C07289=1017.873,162.387,378.674,167.472,52.697,159.777
C07290=1017.878,162.636,378.653,167.475,52.688,159.776
C07291=1017.882,162.885,378.632,167.480,52.680,159.775
C07292=1017.887,163.133,378.611,167.483,52.671,159.774
C07293=1017.892,163.383,378.590,167.486,52.662,159.772
C07294=1017.897,163.632,378.569,167.490,52.654,159.772
C07295=1017.902,163.881,378.548,167.494,52.645,159.771
C07296=1017.906,164.131,378.527,167.498,52.637,159.770
C07297=1017.911,164.379,378.507,167.501,52.628,159.768
C07298=1017.916,164.628,378.485,167.504,52.619,159.767
C07299=1017.921,164.877,378.465,167.508,52.611,159.766
C07300=1017.925,165.127,378.443,167.512,52.602,159.765
C07301=1017.930,165.376,378.422,167.516,52.593,159.764
C07302=1017.935,165.625,378.402,167.519,52.585,159.763
C07303=1017.939,165.873,378.380,167.523,52.575,159.762
C07304=1017.945,166.122,378.360,167.527,52.567,159.761
C07305=1017.949,166.372,378.338,167.530,52.558,159.760
C07306=1017.954,166.621,378.317,167.534,52.550,159.759
C07307=1017.959,166.870,378.296,167.538,52.541,159.758
C07308=1017.964,167.119,378.275,167.542,52.532,159.757
C07309=1017.969,167.368,378.254,167.545,52.524,159.756
C07310=1017.974,167.618,378.233,167.548,52.515,159.755
C07311=1017.978,167.866,378.212,167.553,52.506,159.754
C07312=1017.983,168.115,378.191,167.556,52.498,159.753
C07313=1017.988,168.364,378.170,167.560,52.489,159.752
C07314=1017.993,168.613,378.149,167.564,52.480,159.751
C07315=1017.998,168.862,378.128,167.568,52.472,159.750
C07316=1018.002,169.112,378.106,167.571,52.463,159.749
C07317=1018.008,169.360,378.085,167.575,52.454,159.748
C07318=1018.012,169.610,378.064,167.579,52.446,159.747
C07319=1018.017,169.859,378.043,167.582,52.437,159.746
C07320=1018.022,170.108,378.022,167.587,52.429,159.745
C07321=1018.027,170.357,378.000,167.590,52.420,159.744
C07322=1018.032,170.606,377.980,167.594,52.411,159.743
C07323=1018.038,170.887,377.956,167.598,52.401,159.742
C07324=1018.043,171.168,377.932,167.603,52.392,159.741
C07325=1018.048,171.449,377.908,167.607,52.382,159.739
C07326=1018.054,171.731,377.884,167.611,52.372,159.738
C07327=1018.058,171.980,377.863,167.615,52.364,159.737
C07328=1018.064,172.228,377.842,167.618,52.355,159.736
C07329=1018.069,172.478,377.820,167.623,52.346,159.735
C07330=1018.074,172.727,377.799,167.627,52.338,159.734
C07331=1018.079,172.976,377.778,167.630,52.329,159.733
C07332=1018.084,173.225,377.756,167.634,52.320,159.732
C07333=1018.089,173.474,377.735,167.638,52.312,159.731
C07334=1018.094,173.723,377.713,167.642,52.302,159.730
C07335=1018.098,173.972,377.692,167.645,52.294,159.729
C07336=1018.104,174.221,377.671,167.649,52.286,159.728
C07337=1018.108,174.470,377.650,167.654,52.276,159.727
C07338=1018.114,174.719,377.629,167.657,52.268,159.726
C07339=1018.118,174.968,377.607,167.662,52.259,159.725
C07340=1018.123,175.217,377.586,167.665,52.250,159.724
C07341=1018.129,175.466,377.565,167.669,52.241,159.723
C07342=1018.133,175.715,377.543,167.673,52.233,159.722
C07343=1018.138,175.964,377.522,167.676,52.225,159.721
C07344=1018.143,176.213,377.501,167.681,52.215,159.720
C07345=1018.148,176.462,377.479,167.684,52.207,159.719
C07346=1018.154,176.711,377.458,167.689,52.198,159.718
C07347=1018.159,176.960,377.436,167.692,52.190,159.717
C07348=1018.163,177.210,377.415,167.697,52.181,159.716
C07349=1018.169,177.458,377.394,167.700,52.172,159.715
C07350=1018.174,177.707,377.372,167.705,52.164,159.714
C07351=1018.178,177.956,377.351,167.708,52.155,159.713
C07352=1018.184,178.205,377.329,167.713,52.146,159.712
C07353=1018.189,178.454,377.307,167.716,52.138,159.711
C07354=1018.194,178.704,377.286,167.721,52.129,159.710
C07355=1018.199,178.952,377.265,167.724,52.120,159.709
C07356=1018.204,179.201,377.243,167.729,52.112,159.708
C07357=1018.210,179.450,377.222,167.732,52.103,159.707
C07358=1018.214,179.699,377.200,167.737,52.094,159.706
C07359=1018.220,179.949,377.178,167.740,52.086,159.705
C07360=1018.225,180.198,377.158,167.745,52.077,159.704
C07361=1018.230,180.447,377.136,167.748,52.068,159.703
C07362=1018.235,180.695,377.114,167.753,52.060,159.702
C07363=1018.240,180.944,377.093,167.756,52.051,159.701
C07364=1018.245,181.194,377.071,167.761,52.042,159.700
C07365=1018.250,181.443,377.049,167.764,52.034,159.699
C07366=1018.256,181.691,377.028,167.769,52.025,159.698
C07367=1018.261,181.940,377.006,167.772,52.016,159.697
C07368=1018.266,182.190,376.984,167.777,52.008,159.696
C07369=1018.270,182.439,376.961,167.781,52.000,159.695
C07370=1018.275,182.688,376.940,167.785,51.991,159.694
C07371=1018.280,182.937,376.918,167.789,51.983,159.693
C07372=1018.284,183.186,376.895,167.793,51.975,159.692
C07373=1018.289,183.435,376.873,167.797,51.965,159.691
C07374=1018.294,183.684,376.851,167.801,51.957,159.690
C07375=1018.299,183.933,376.829,167.805,51.949,159.689
C07376=1018.303,184.182,376.807,167.809,51.941,159.688
C07377=1018.309,184.431,376.784,167.813,51.932,159.687
C07378=1018.314,184.680,376.762,167.818,51.924,159.686
C07379=1018.318,184.928,376.740,167.821,51.916,159.685
C07380=1018.322,185.178,376.718,167.825,51.907,159.684
C07381=1018.328,185.427,376.695,167.830,51.899,159.684
C07382=1018.333,185.675,376.673,167.833,51.891,159.683
C07383=1018.337,185.924,376.650,167.838,51.882,159.682
C07384=1018.342,186.173,376.629,167.842,51.874,159.681
C07385=1018.347,186.423,376.606,167.846,51.865,159.680
C07386=1018.351,186.672,376.584,167.850,51.857,159.679
C07387=1018.357,186.952,376.559,167.854,51.848,159.678
C07388=1018.363,187.233,376.533,167.860,51.838,159.677
C07389=1018.368,187.514,376.508,167.864,51.829,159.676
C07390=1018.374,187.794,376.483,167.869,51.819,159.675
C07391=1018.379,188.044,376.461,167.872,51.811,159.674
C07392=1018.384,188.292,376.439,167.877,51.802,159.673
C07393=1018.388,188.541,376.416,167.881,51.794,159.672
C07394=1018.394,188.790,376.393,167.886,51.785,159.671
C07395=1018.398,189.039,376.371,167.889,51.777,159.670
C07396=1018.403,189.288,376.348,167.894,51.769,159.669
C07397=1018.408,189.537,376.326,167.898,51.761,159.668
C07398=1018.413,189.786,376.304,167.903,51.752,159.667
C07399=1018.419,190.035,376.281,167.906,51.744,159.666
C07400=1018.423,190.284,376.259,167.911,51.736,159.665
C07401=1018.428,190.533,376.237,167.915,51.727,159.664
C07402=1018.433,190.782,376.214,167.919,51.719,159.663
C07403=1018.438,191.031,376.192,167.923,51.711,159.662
C07404=1018.443,191.280,376.169,167.928,51.702,159.661
C07405=1018.448,191.529,376.147,167.932,51.694,159.661
C07406=1018.453,191.777,376.124,167.936,51.685,159.660
C07407=1018.458,192.027,376.101,167.940,51.677,159.659
C07408=1018.463,192.275,376.079,167.945,51.668,159.658
C07409=1018.468,192.525,376.056,167.949,51.660,159.657
C07410=1018.473,192.773,376.034,167.953,51.651,159.656
C07411=1018.478,193.022,376.011,167.958,51.643,159.655
C07412=1018.483,193.271,375.989,167.962,51.635,159.654
C07413=1018.488,193.520,375.966,167.967,51.627,159.653
C07414=1018.493,193.769,375.944,167.970,51.618,159.652
C07415=1018.498,194.017,375.921,167.975,51.610,159.651
C07416=1018.503,194.267,375.898,167.980,51.602,159.651
C07417=1018.508,194.515,375.876,167.983,51.593,159.649
C07418=1018.514,194.764,375.853,167.988,51.585,159.649
C07419=1018.518,195.014,375.830,167.992,51.577,159.648
C07420=1018.523,195.262,375.808,167.996,51.568,159.647
C07421=1018.529,195.512,375.785,168.001,51.559,159.646
C07422=1018.533,195.760,375.762,168.005,51.551,159.645
C07423=1018.539,196.009,375.739,168.010,51.543,159.644
C07424=1018.544,196.258,375.717,168.013,51.535,159.643
C07425=1018.549,196.507,375.694,168.018,51.526,159.642
C07426=1018.554,196.756,375.672,168.023,51.518,159.641
C07427=1018.559,197.005,375.649,168.027,51.509,159.640
C07428=1018.564,197.253,375.626,168.032,51.501,159.639
C07429=1018.569,197.503,375.604,168.036,51.493,159.639
C07430=1018.575,197.752,375.581,168.040,51.485,159.638
C07431=1018.580,198.000,375.558,168.045,51.476,159.637
C07432=1018.585,198.249,375.534,168.050,51.468,159.636
C07433=1018.590,198.498,375.513,168.054,51.460,159.635
C07434=1018.596,198.747,375.490,168.058,51.451,159.634
C07435=1018.601,198.996,375.466,168.063,51.442,159.633
C07436=1018.605,199.245,375.444,168.068,51.434,159.632
C07437=1018.610,199.494,375.421,168.072,51.426,159.631
C07438=1018.616,199.743,375.398,168.077,51.418,159.630
C07439=1018.621,199.992,375.375,168.081,51.410,159.630
C07440=1018.625,200.241,375.351,168.085,51.402,159.629
C07441=1018.631,200.490,375.328,168.090,51.393,159.628
C07442=1018.636,200.738,375.305,168.094,51.385,159.627
C07443=1018.641,200.987,375.281,168.099,51.377,159.626
C07444=1018.645,201.236,375.258,168.103,51.369,159.625
C07445=1018.651,201.485,375.235,168.108,51.361,159.624
C07446=1018.656,201.734,375.212,168.112,51.352,159.623
C07447=1018.660,201.983,375.189,168.116,51.344,159.622
C07448=1018.666,202.231,375.166,168.121,51.336,159.622
C07449=1018.671,202.481,375.142,168.126,51.328,159.621
C07450=1018.675,202.729,375.119,168.130,51.320,159.620
C07451=1018.702,203.979,375.000,168.600,51.411,159.725
C07452=1018.707,204.207,374.977,168.603,51.404,159.724
C07453=1018.713,204.434,374.955,168.607,51.398,159.723
C07454=1018.718,204.661,374.932,168.610,51.391,159.723
C07455=1018.724,204.888,374.910,168.614,51.385,159.722
C07456=1018.730,205.116,374.887,168.617,51.378,159.721
C07457=1018.735,205.343,374.863,168.620,51.372,159.720
C07458=1018.740,205.570,374.841,168.624,51.365,159.720
C07459=1018.747,205.819,374.816,168.628,51.358,159.719
C07460=1018.753,206.068,374.791,168.631,51.351,159.718
C07461=1018.758,206.316,374.766,168.635,51.343,159.717
C07462=1018.764,206.565,374.741,168.640,51.336,159.716
C07463=1018.771,206.813,374.716,168.643,51.329,159.715
C07464=1018.777,207.062,374.690,168.647,51.322,159.715
C07465=1018.782,207.311,374.666,168.650,51.315,159.714
C07466=1018.788,207.559,374.641,168.655,51.308,159.713
C07467=1018.794,207.808,374.615,168.658,51.301,159.712
C07468=1018.801,208.057,374.590,168.662,51.294,159.711
C07469=1018.806,208.305,374.565,168.666,51.287,159.711
C07470=1018.812,208.554,374.540,168.670,51.280,159.710
C07471=1018.818,208.803,374.515,168.674,51.273,159.709
C07472=1018.824,209.052,374.489,168.677,51.266,159.708
C07473=1018.830,209.300,374.464,168.682,51.260,159.707
C07474=1018.836,209.548,374.439,168.685,51.253,159.707
C07475=1018.842,209.797,374.414,168.689,51.246,159.706
C07476=1018.848,210.046,374.388,168.692,51.239,159.705
C07477=1018.854,210.294,374.363,168.697,51.232,159.704
C07478=1018.860,210.543,374.337,168.700,51.225,159.703
C07479=1018.866,210.792,374.312,168.705,51.218,159.703
C07480=1018.872,211.040,374.287,168.708,51.212,159.702
C07481=1018.878,211.289,374.261,168.712,51.204,159.701
C07482=1018.883,211.538,374.235,168.715,51.198,159.700
C07483=1018.889,211.786,374.210,168.720,51.191,159.700
C07484=1018.896,212.035,374.185,168.723,51.184,159.699
C07485=1018.901,212.284,374.159,168.728,51.177,159.698
C07486=1018.907,212.533,374.133,168.731,51.170,159.697
C07487=1018.913,212.781,374.108,168.735,51.164,159.696
C07488=1018.919,213.029,374.083,168.739,51.157,159.696
C07489=1018.925,213.278,374.057,168.742,51.150,159.695
C07490=1018.931,213.527,374.032,168.747,51.144,159.694
C07491=1018.937,213.775,374.006,168.750,51.137,159.693
C07492=1018.942,214.024,373.981,168.754,51.130,159.693
C07493=1018.949,214.273,373.955,168.758,51.124,159.692
C07494=1018.955,214.521,373.929,168.762,51.117,159.691
C07495=1018.961,214.770,373.904,168.765,51.110,159.690
C07496=1018.967,215.019,373.878,168.770,51.103,159.690
C07497=1018.973,215.268,373.853,168.773,51.096,159.689
C07498=1018.979,215.516,373.827,168.777,51.090,159.688
C07499=1018.984,215.764,373.802,168.781,51.083,159.687
C07500=1018.990,216.013,373.776,168.785,51.076,159.687
C07501=1018.997,216.261,373.750,168.789,51.070,159.686
C07502=1019.003,216.510,373.725,168.793,51.063,159.685
C07503=1019.009,216.759,373.699,168.797,51.057,159.685
C07504=1019.015,217.007,373.674,168.801,51.050,159.684
C07505=1019.021,217.256,373.648,168.805,51.043,159.683
C07506=1019.027,217.505,373.622,168.809,51.037,159.682
C07507=1019.033,217.753,373.596,168.812,51.031,159.682
C07508=1019.039,218.002,373.571,168.816,51.023,159.681
C07509=1019.046,218.250,373.545,168.820,51.017,159.680
C07510=1019.051,218.499,373.519,168.824,51.010,159.679
C07511=1019.057,218.726,373.495,168.827,51.004,159.679
C07512=1019.062,218.955,373.472,168.831,50.999,159.678
C07513=1019.068,219.183,373.448,168.835,50.993,159.677
C07514=1019.073,219.411,373.423,168.839,50.987,159.677
C07515=1019.078,219.639,373.400,168.842,50.981,159.676
C07516=1019.084,219.867,373.376,168.846,50.975,159.676
C07517=1019.089,220.095,373.352,168.849,50.969,159.675
C07518=1019.095,220.322,373.328,168.853,50.963,159.674
C07519=1019.100,220.571,373.302,168.856,50.957,159.674
C07520=1019.107,220.819,373.276,168.861,50.950,159.673
C07521=1019.112,221.068,373.250,168.864,50.944,159.672
C07522=1019.118,221.317,373.223,168.868,50.938,159.671
C07523=1019.124,221.565,373.198,168.873,50.931,159.671
C07524=1019.131,221.814,373.171,168.876,50.925,159.670
C07525=1019.137,222.063,373.146,168.880,50.919,159.669
C07526=1019.143,222.311,373.119,168.884,50.912,159.669
C07527=1019.148,222.560,373.093,168.888,50.906,159.668
C07528=1019.155,222.808,373.067,168.892,50.900,159.667
C07529=1019.160,223.057,373.041,168.897,50.894,159.667
C07530=1019.167,223.305,373.015,168.900,50.887,159.666
C07531=1019.172,223.554,372.988,168.904,50.881,159.665
C07532=1019.178,223.803,372.962,168.908,50.874,159.665
C07533=1019.185,224.052,372.936,168.912,50.868,159.664
C07534=1019.190,224.300,372.910,168.916,50.862,159.663
C07535=1019.197,224.549,372.884,168.920,50.856,159.663
C07536=1019.203,224.797,372.857,168.924,50.850,159.662
C07537=1019.208,225.046,372.832,168.928,50.843,159.662
C07538=1019.215,225.294,372.805,168.932,50.836,159.661
C07539=1019.220,225.542,372.779,168.936,50.830,159.660
C07540=1019.227,225.792,372.753,168.940,50.824,159.659
C07541=1019.233,226.040,372.726,168.944,50.818,159.659
C07542=1019.239,226.288,372.700,168.948,50.812,159.658
C07543=1019.245,226.536,372.674,168.952,50.806,159.658
C07544=1019.251,226.785,372.648,168.955,50.800,159.657
C07545=1019.257,227.034,372.621,168.960,50.793,159.656
C07546=1019.263,227.283,372.594,168.964,50.787,159.656
C07547=1019.269,227.531,372.568,168.967,50.781,159.655
C07548=1019.275,227.779,372.541,168.972,50.776,159.655
C07549=1019.281,228.028,372.515,168.976,50.769,159.654
C07550=1019.287,228.276,372.488,168.980,50.763,159.653
C07551=1019.293,228.526,372.462,168.984,50.757,159.653
C07552=1019.299,228.774,372.435,168.987,50.751,159.652
C07553=1019.305,229.022,372.409,168.992,50.745,159.651
C07554=1019.311,229.270,372.383,168.996,50.738,159.651
C07555=1019.317,229.519,372.355,169.000,50.733,159.650
C07556=1019.323,229.768,372.329,169.004,50.727,159.650
C07557=1019.329,230.016,372.302,169.007,50.721,159.649
C07558=1019.335,230.265,372.276,169.012,50.715,159.648
C07559=1019.341,230.514,372.249,169.016,50.709,159.648
C07560=1019.347,230.762,372.222,169.020,50.703,159.647
C07561=1019.353,231.010,372.195,169.024,50.697,159.647
C07562=1019.358,231.259,372.169,169.028,50.692,159.646
C07563=1019.365,231.508,372.142,169.033,50.685,159.646
C07564=1019.371,231.755,372.114,169.036,50.679,159.645
C07565=1019.377,232.004,372.088,169.040,50.674,159.644
C07566=1019.383,232.253,372.061,169.044,50.668,159.644
C07567=1019.389,232.501,372.034,169.048,50.662,159.643
C07568=1019.394,232.750,372.007,169.053,50.656,159.643
C07569=1019.400,232.998,371.981,169.057,50.650,159.642
C07570=1019.407,233.247,371.954,169.060,50.644,159.641
C07571=1019.412,233.470,371.929,169.064,50.639,159.641
C07572=1019.418,233.695,371.905,169.068,50.633,159.640
C07573=1019.423,233.918,371.881,169.072,50.628,159.640
C07574=1019.429,234.143,371.857,169.075,50.623,159.639
C07575=1019.434,234.366,371.833,169.079,50.618,159.639
C07576=1019.440,234.590,371.808,169.082,50.613,159.638
C07577=1019.445,234.814,371.784,169.086,50.607,159.638
C07578=1019.450,235.038,371.759,169.089,50.602,159.637
C07579=1019.456,235.286,371.732,169.094,50.596,159.637
C07580=1019.462,235.534,371.706,169.098,50.590,159.636
C07581=1019.468,235.783,371.678,169.102,50.585,159.636
C07582=1019.474,236.031,371.651,169.106,50.579,159.635
C07583=1019.481,236.280,371.624,169.110,50.574,159.635
C07584=1019.487,236.528,371.597,169.114,50.568,159.634
C07585=1019.492,236.776,371.570,169.119,50.562,159.634
C07586=1019.499,237.025,371.543,169.123,50.556,159.633
C07587=1019.505,237.273,371.516,169.127,50.551,159.632
C07588=1019.511,237.522,371.489,169.131,50.545,159.632
C07589=1019.517,237.771,371.462,169.135,50.539,159.631
C07590=1019.524,238.019,371.434,169.139,50.534,159.631
C07591=1019.529,238.267,371.408,169.144,50.527,159.630
C07592=1019.535,238.516,371.381,169.148,50.522,159.630
C07593=1019.541,238.765,371.353,169.152,50.517,159.629
C07594=1019.547,239.013,371.326,169.156,50.511,159.629
C07595=1019.554,239.261,371.298,169.160,50.505,159.628
C07596=1019.559,239.510,371.272,169.164,50.500,159.628
C07597=1019.565,239.758,371.244,169.168,50.495,159.627
C07598=1019.571,240.007,371.217,169.172,50.489,159.627
C07599=1019.578,240.255,371.189,169.176,50.483,159.626
C07600=1019.583,240.503,371.161,169.180,50.478,159.626
C07601=1019.590,240.752,371.134,169.185,50.472,159.625
C07602=1019.596,241.000,371.107,169.189,50.467,159.625
C07603=1019.602,241.249,371.078,169.194,50.461,159.624
C07604=1019.607,241.497,371.052,169.197,50.455,159.624
C07605=1019.614,241.746,371.024,169.201,50.450,159.623
C07606=1019.619,241.994,370.996,169.206,50.445,159.623
C07607=1019.626,242.243,370.969,169.210,50.439,159.622
C07608=1019.632,242.491,370.942,169.214,50.434,159.622
C07609=1019.638,242.739,370.913,169.218,50.429,159.621
C07610=1019.644,242.988,370.887,169.222,50.423,159.621
C07611=1019.650,243.236,370.859,169.226,50.418,159.620
C07612=1019.656,243.484,370.831,169.230,50.413,159.620
C07613=1019.661,243.733,370.803,169.235,50.407,159.620
C07614=1019.668,243.981,370.775,169.239,50.402,159.619
C07615=1019.673,244.230,370.748,169.243,50.397,159.619
C07616=1019.679,244.478,370.720,169.247,50.391,159.618
C07617=1019.685,244.726,370.692,169.251,50.386,159.618
C07618=1019.691,244.975,370.664,169.255,50.381,159.617
C07619=1019.697,245.223,370.636,169.259,50.375,159.617
C07620=1019.703,245.472,370.608,169.264,50.370,159.616
C07621=1019.709,245.720,370.580,169.268,50.365,159.616
C07622=1019.715,245.968,370.552,169.272,50.360,159.616
C07623=1019.721,246.217,370.524,169.276,50.355,159.615
C07624=1019.726,246.465,370.496,169.280,50.349,159.615
C07625=1019.733,246.713,370.468,169.285,50.344,159.614
C07626=1019.739,246.962,370.440,169.289,50.339,159.614
C07627=1019.744,247.210,370.412,169.293,50.334,159.613
C07628=1019.751,247.459,370.384,169.297,50.329,159.613
C07629=1019.756,247.707,370.356,169.302,50.323,159.612
C07630=1019.762,247.956,370.328,169.307,50.318,159.612
C07631=1019.768,248.176,370.304,169.310,50.313,159.612
C07632=1019.773,248.397,370.278,169.314,50.309,159.611
C07633=1019.779,248.617,370.254,169.318,50.304,159.611
C07634=1019.784,248.838,370.229,169.321,50.299,159.610
C07635=1019.790,249.059,370.204,169.325,50.295,159.610
C07636=1019.794,249.279,370.179,169.330,50.290,159.610
C07637=1019.801,249.500,370.154,169.333,50.286,159.610
C07638=1019.805,249.721,370.129,169.337,50.282,159.609
C07639=1019.812,249.968,370.101,169.341,50.276,159.609
C07640=1019.818,250.216,370.073,169.345,50.271,159.608
C07641=1019.824,250.465,370.044,169.349,50.266,159.608
C07642=1019.830,250.714,370.017,169.354,50.261,159.607
C07643=1019.836,250.962,369.988,169.358,50.256,159.607
C07644=1019.842,251.210,369.960,169.362,50.251,159.607
C07645=1019.849,251.458,369.932,169.366,50.246,159.606
C07646=1019.854,251.707,369.904,169.371,50.240,159.606
C07647=1019.860,251.956,369.875,169.375,50.236,159.606
C07648=1019.867,252.204,369.848,169.379,50.230,159.605
C07649=1019.873,252.452,369.819,169.384,50.226,159.605
C07650=1019.879,252.700,369.790,169.388,50.220,159.604
C07651=1019.885,252.949,369.763,169.392,50.215,159.604
C07652=1019.891,253.198,369.734,169.397,50.210,159.604
C07653=1019.897,253.445,369.706,169.401,50.205,159.603
C07654=1019.904,253.694,369.678,169.405,50.200,159.603
C07655=1019.910,253.942,369.650,169.410,50.195,159.602
C07656=1019.916,254.190,369.621,169.414,50.191,159.602
C07657=1019.923,254.439,369.593,169.418,50.185,159.602
C07658=1019.928,254.688,369.565,169.423,50.181,159.601
C07659=1019.934,254.935,369.536,169.427,50.175,159.601
C07660=1019.941,255.183,369.508,169.431,50.171,159.601
C07661=1019.947,255.432,369.480,169.436,50.165,159.600
C07662=1019.953,255.680,369.451,169.440,50.161,159.600
C07663=1019.960,255.929,369.423,169.444,50.155,159.599
C07664=1019.966,256.177,369.394,169.449,50.151,159.599
C07665=1019.972,256.426,369.366,169.453,50.145,159.599
C07666=1019.979,256.673,369.337,169.458,50.141,159.598
C07667=1019.985,256.922,369.309,169.462,50.136,159.598
C07668=1019.990,257.170,369.281,169.467,50.131,159.598
C07669=1019.997,257.418,369.253,169.472,50.126,159.597
C07670=1020.003,257.667,369.224,169.476,50.121,159.597
C07671=1020.009,257.915,369.195,169.481,50.116,159.597
C07672=1020.016,258.163,369.167,169.485,50.111,159.596
C07673=1020.022,258.412,369.138,169.489,50.106,159.596
C07674=1020.029,258.660,369.109,169.494,50.101,159.596
C07675=1020.035,258.908,369.082,169.498,50.097,159.595
C07676=1020.041,259.156,369.053,169.503,50.091,159.595
C07677=1020.047,259.405,369.024,169.507,50.087,159.595
C07678=1020.054,259.653,368.996,169.512,50.082,159.594
C07679=1020.060,259.902,368.968,169.516,50.077,159.594
C07680=1020.067,260.150,368.938,169.520,50.072,159.594
C07681=1020.073,260.398,368.909,169.525,50.068,159.593
C07682=1020.079,260.646,368.880,169.529,50.063,159.593
C07683=1020.085,260.894,368.851,169.533,50.059,159.593
C07684=1020.091,261.143,368.823,169.538,50.054,159.592
C07685=1020.097,261.391,368.794,169.542,50.049,159.592
C07686=1020.104,261.639,368.765,169.547,50.045,159.592
C07687=1020.110,261.887,368.736,169.551,50.040,159.592
C07688=1020.116,262.135,368.707,169.556,50.036,159.591
C07689=1020.122,262.384,368.677,169.560,50.031,159.591
C07690=1020.128,262.632,368.648,169.565,50.026,159.591
C07691=1020.134,262.852,368.623,169.568,50.022,159.590
C07692=1020.139,263.071,368.597,169.572,50.018,159.590
C07693=1020.144,263.291,368.572,169.577,50.014,159.590
C07694=1020.150,263.512,368.546,169.580,50.010,159.590
C07695=1020.156,263.731,368.520,169.584,50.006,159.589
C07696=1020.161,263.951,368.494,169.588,50.002,159.589
C07697=1020.167,264.170,368.469,169.593,49.998,159.589
C07698=1020.172,264.390,368.443,169.596,49.993,159.589
C07699=1020.178,264.638,368.414,169.601,49.989,159.589
C07700=1020.184,264.887,368.385,169.606,49.985,159.588
C07701=1020.190,265.135,368.356,169.610,49.980,159.588
C07702=1020.197,265.384,368.326,169.615,49.976,159.588
C07703=1020.204,265.631,368.297,169.620,49.971,159.587
C07704=1020.209,265.880,368.267,169.624,49.966,159.587
C07705=1020.216,266.128,368.238,169.628,49.962,159.587
C07706=1020.222,266.376,368.209,169.633,49.958,159.587
C07707=1020.228,266.624,368.180,169.637,49.953,159.586
C07708=1020.234,266.872,368.150,169.642,49.949,159.586
C07709=1020.240,267.120,368.120,169.646,49.944,159.586
C07710=1020.247,267.369,368.091,169.651,49.940,159.586
C07711=1020.253,267.617,368.062,169.656,49.936,159.585
C07712=1020.259,267.865,368.032,169.660,49.931,159.585
C07713=1020.265,268.113,368.003,169.665,49.926,159.585
C07714=1020.272,268.361,367.974,169.670,49.923,159.585
C07715=1020.277,268.609,367.944,169.674,49.918,159.585
C07716=1020.284,268.858,367.915,169.678,49.914,159.584
C07717=1020.291,269.106,367.885,169.683,49.910,159.584
C07718=1020.297,269.354,367.856,169.687,49.905,159.584
C07719=1020.302,269.602,367.826,169.692,49.901,159.584
C07720=1020.309,269.850,367.796,169.697,49.897,159.583
C07721=1020.315,270.099,367.766,169.701,49.892,159.583
C07722=1020.322,270.346,367.737,169.706,49.888,159.583
C07723=1020.328,270.595,367.708,169.711,49.883,159.583
C07724=1020.333,270.843,367.678,169.716,49.879,159.583
C07725=1020.340,271.091,367.648,169.719,49.875,159.582
C07726=1020.346,271.340,367.618,169.724,49.871,159.582
C07727=1020.353,271.587,367.588,169.729,49.867,159.582
C07728=1020.358,271.836,367.559,169.733,49.862,159.582
C07729=1020.365,272.084,367.529,169.738,49.858,159.582
C07730=1020.371,272.332,367.500,169.743,49.854,159.581
C07731=1020.377,272.580,367.469,169.748,49.850,159.581
C07732=1020.384,272.828,367.439,169.753,49.846,159.581
C07733=1020.390,273.076,367.409,169.757,49.841,159.581
C07734=1020.396,273.324,367.380,169.761,49.837,159.581
C07735=1020.402,273.572,367.350,169.766,49.833,159.580
C07736=1020.409,273.821,367.320,169.771,49.829,159.580
C07737=1020.415,274.068,367.290,169.776,49.825,159.580
C07738=1020.421,274.317,367.261,169.780,49.820,159.580
C07739=1020.428,274.565,367.230,169.785,49.816,159.580
C07740=1020.434,274.813,367.200,169.790,49.813,159.580
C07741=1020.440,275.060,367.170,169.795,49.808,159.580
C07742=1020.446,275.310,367.140,169.800,49.804,159.579
C07743=1020.453,275.557,367.110,169.804,49.800,159.579
C07744=1020.459,275.806,367.079,169.808,49.796,159.579
C07745=1020.466,276.053,367.050,169.813,49.792,159.579
C07746=1020.471,276.302,367.020,169.818,49.788,159.579
C07747=1020.478,276.550,366.990,169.823,49.784,159.579
C07748=1020.484,276.798,366.959,169.828,49.779,159.578
C07749=1020.491,277.046,366.929,169.833,49.776,159.578
C07750=1020.497,277.294,366.899,169.838,49.772,159.578
C07751=1020.503,277.515,366.872,169.841,49.768,159.578
C07752=1020.508,277.739,366.845,169.845,49.764,159.578
C07753=1020.513,277.960,366.817,169.850,49.761,159.578
C07754=1020.519,278.182,366.790,169.855,49.758,159.578
C07755=1020.525,278.404,366.763,169.859,49.754,159.578
C07756=1020.530,278.626,366.736,169.862,49.750,159.577
C07757=1020.536,278.849,366.709,169.867,49.747,159.578
C07758=1020.541,279.071,366.681,169.872,49.743,159.577
C07759=1020.548,279.319,366.651,169.876,49.740,159.577
C07760=1020.554,279.567,366.621,169.881,49.736,159.577
C07761=1020.560,279.815,366.591,169.886,49.732,159.577
C07762=1020.567,280.063,366.559,169.890,49.728,159.577
C07763=1020.572,280.310,366.529,169.895,49.724,159.577
C07764=1020.580,280.559,366.499,169.900,49.720,159.577
C07765=1020.585,280.806,366.468,169.905,49.716,159.577
C07766=1020.592,281.055,366.438,169.910,49.712,159.577
C07767=1020.598,281.303,366.407,169.914,49.709,159.576
C07768=1020.605,281.551,366.377,169.919,49.705,159.576
C07769=1020.611,281.799,366.346,169.924,49.701,159.576
C07770=1020.617,282.047,366.315,169.929,49.697,159.576
C07771=1020.624,282.295,366.285,169.934,49.693,159.576
C07772=1020.630,282.543,366.254,169.939,49.689,159.576
C07773=1020.637,282.791,366.224,169.944,49.685,159.576
C07774=1020.643,283.039,366.193,169.949,49.682,159.576
C07775=1020.649,283.287,366.162,169.953,49.679,159.576
C07776=1020.656,283.535,366.132,169.958,49.675,159.576
C07777=1020.661,283.783,366.101,169.963,49.671,159.576
C07778=1020.669,284.031,366.071,169.968,49.667,159.576
C07779=1020.675,284.279,366.040,169.973,49.663,159.575
C07780=1020.681,284.527,366.009,169.978,49.660,159.576
C07781=1020.688,284.775,365.978,169.983,49.656,159.575
C07782=1020.694,285.023,365.948,169.988,49.652,159.575
C07783=1020.701,285.271,365.917,169.993,49.648,159.575
C07784=1020.708,285.519,365.886,169.997,49.645,159.575
C07785=1020.714,285.766,365.855,170.002,49.641,159.575
C07786=1020.720,286.015,365.824,170.007,49.637,159.575
C07787=1020.726,286.263,365.792,170.013,49.634,159.575
C07788=1020.732,286.511,365.762,170.017,49.630,159.575
C07789=1020.739,286.759,365.731,170.022,49.626,159.575
C07790=1020.745,287.007,365.700,170.028,49.623,159.575
C07791=1020.751,287.254,365.669,170.032,49.619,159.575
C07792=1020.758,287.503,365.638,170.037,49.616,159.575
C07793=1020.764,287.751,365.607,170.042,49.612,159.575
C07794=1020.771,287.999,365.575,170.047,49.608,159.575
C07795=1020.777,288.247,365.545,170.052,49.605,159.575
C07796=1020.784,288.494,365.513,170.057,49.601,159.575
C07797=1020.790,288.742,365.482,170.062,49.598,159.575
C07798=1020.797,288.990,365.450,170.067,49.594,159.575
C07799=1020.803,289.238,365.420,170.072,49.591,159.575
C07800=1020.810,289.486,365.389,170.077,49.588,159.575
C07801=1020.816,289.734,365.357,170.082,49.584,159.575
C07802=1020.823,289.982,365.326,170.087,49.581,159.575
C07803=1020.828,290.230,365.295,170.092,49.577,159.575
C07804=1020.835,290.478,365.263,170.098,49.573,159.575
C07805=1020.842,290.726,365.232,170.102,49.569,159.575
C07806=1020.848,290.974,365.201,170.108,49.566,159.575
C07807=1020.855,291.222,365.169,170.112,49.563,159.575
C07808=1020.861,291.470,365.138,170.117,49.559,159.575
C07809=1020.868,291.717,365.107,170.122,49.556,159.575
C07810=1020.874,291.966,365.075,170.128,49.553,159.575
C07811=1020.881,292.193,365.046,170.132,49.550,159.575
C07812=1020.886,292.421,365.018,170.137,49.546,159.575
C07813=1020.892,292.650,364.989,170.141,49.543,159.575
C07814=1020.898,292.878,364.959,170.147,49.540,159.575
C07815=1020.904,293.106,364.931,170.151,49.537,159.575
C07816=1020.910,293.334,364.901,170.155,49.534,159.575
C07817=1020.916,293.563,364.872,170.160,49.531,159.575
C07818=1020.922,293.790,364.843,170.165,49.528,159.575
C07819=1020.928,294.039,364.811,170.170,49.525,159.575
C07820=1020.934,294.287,364.779,170.175,49.521,159.576
C07821=1020.940,294.535,364.747,170.181,49.518,159.576
C07822=1020.947,294.782,364.715,170.186,49.515,159.576
C07823=1020.953,295.030,364.683,170.190,49.512,159.576
C07824=1020.959,295.279,364.651,170.196,49.509,159.576
C07825=1020.965,295.526,364.620,170.201,49.506,159.576
C07826=1020.972,295.773,364.587,170.206,49.502,159.576
C07827=1020.978,296.022,364.555,170.212,49.499,159.576
C07828=1020.985,296.269,364.524,170.217,49.496,159.576
C07829=1020.991,296.517,364.491,170.221,49.493,159.576
C07830=1020.998,296.765,364.460,170.227,49.490,159.576
C07831=1021.004,297.013,364.427,170.232,49.486,159.576
C07832=1021.010,297.261,364.395,170.237,49.483,159.577
C07833=1021.017,297.509,364.363,170.242,49.480,159.577
C07834=1021.023,297.756,364.331,170.248,49.477,159.577
C07835=1021.030,298.004,364.299,170.252,49.474,159.577
C07836=1021.036,298.252,364.267,170.258,49.471,159.577
C07837=1021.043,298.500,364.235,170.263,49.468,159.577
C07838=1021.049,298.747,364.202,170.268,49.465,159.577
C07839=1021.055,298.995,364.170,170.274,49.462,159.577
C07840=1021.062,299.243,364.138,170.279,49.458,159.577
C07841=1021.068,299.491,364.106,170.284,49.455,159.578
C07842=1021.075,299.738,364.074,170.290,49.452,159.578
C07843=1021.081,299.986,364.042,170.294,49.450,159.578
C07844=1021.088,300.235,364.009,170.300,49.446,159.578
C07845=1021.095,300.482,363.977,170.305,49.443,159.578
C07846=1021.101,300.730,363.945,170.311,49.441,159.578
C07847=1021.108,300.978,363.913,170.316,49.437,159.578
C07848=1021.114,301.226,363.881,170.321,49.434,159.579
C07849=1021.120,301.473,363.848,170.327,49.431,159.579
C07850=1021.127,301.721,363.816,170.332,49.428,159.579
C07851=1021.133,301.969,363.784,170.338,49.425,159.579
C07852=1021.141,302.217,363.751,170.342,49.422,159.579
C07853=1021.147,302.464,363.718,170.348,49.420,159.579
C07854=1021.153,302.712,363.686,170.353,49.416,159.579
C07855=1021.160,302.960,363.654,170.358,49.413,159.580
C07856=1021.166,303.207,363.621,170.364,49.410,159.580
C07857=1021.174,303.455,363.589,170.369,49.407,159.580
C07858=1021.180,303.703,363.556,170.374,49.404,159.580
C07859=1021.187,303.951,363.523,170.380,49.401,159.580
C07860=1021.193,304.199,363.492,170.385,49.398,159.580
C07861=1021.200,304.447,363.459,170.391,49.396,159.581
C07862=1021.207,304.694,363.427,170.396,49.392,159.581
C07863=1021.214,304.942,363.394,170.402,49.390,159.581
C07864=1021.220,305.189,363.361,170.407,49.387,159.581
C07865=1021.227,305.437,363.329,170.412,49.384,159.581
C07866=1021.234,305.685,363.296,170.417,49.381,159.581
C07867=1021.241,305.932,363.264,170.423,49.379,159.582
C07868=1021.248,306.180,363.231,170.428,49.375,159.582
C07869=1021.254,306.428,363.198,170.434,49.373,159.582
C07870=1021.261,306.675,363.166,170.439,49.370,159.582
C07871=1021.267,306.913,363.135,170.445,49.367,159.582
C07872=1021.274,307.149,363.104,170.450,49.364,159.583
C07873=1021.280,307.386,363.072,170.455,49.361,159.583
C07874=1021.286,307.624,363.041,170.461,49.359,159.583
C07875=1021.294,307.861,363.010,170.466,49.356,159.583
C07876=1021.300,308.098,362.978,170.471,49.353,159.583
C07877=1021.307,308.335,362.947,170.476,49.351,159.584
C07878=1021.313,308.572,362.916,170.482,49.348,159.584
C07879=1021.320,308.820,362.883,170.487,49.345,159.584
C07880=1021.327,309.068,362.850,170.493,49.342,159.584
C07881=1021.334,309.314,362.817,170.499,49.340,159.585
C07882=1021.341,309.563,362.784,170.504,49.337,159.585
C07883=1021.348,309.810,362.752,170.510,49.334,159.585
C07884=1021.354,310.058,362.719,170.515,49.331,159.585
C07885=1021.361,310.305,362.685,170.521,49.329,159.586
C07886=1021.368,310.553,362.652,170.527,49.326,159.586
C07887=1021.375,310.801,362.619,170.532,49.324,159.586
C07888=1021.381,311.048,362.586,170.537,49.322,159.586
C07889=1021.387,311.296,362.551,170.543,49.319,159.587
C07890=1021.394,311.544,362.519,170.548,49.316,159.587
C07891=1021.400,311.791,362.485,170.554,49.314,159.587
C07892=1021.408,312.038,362.451,170.560,49.311,159.587
C07893=1021.413,312.286,362.418,170.565,49.309,159.588
C07894=1021.420,312.534,362.384,170.571,49.306,159.588
C07895=1021.427,312.781,362.351,170.577,49.303,159.588
C07896=1021.434,313.029,362.318,170.583,49.301,159.589
C07897=1021.440,313.277,362.284,170.588,49.298,159.589
C07898=1021.447,313.524,362.250,170.594,49.296,159.589
C07899=1021.453,313.772,362.217,170.599,49.294,159.589
C07900=1021.460,314.019,362.183,170.605,49.292,159.590
C07901=1021.467,314.267,362.149,170.610,49.289,159.590
C07902=1021.473,314.514,362.115,170.616,49.286,159.590
C07903=1021.480,314.763,362.082,170.622,49.284,159.591
C07904=1021.487,315.010,362.049,170.627,49.281,159.591
C07905=1021.493,315.258,362.014,170.633,49.279,159.591
C07906=1021.501,315.505,361.981,170.639,49.277,159.592
C07907=1021.507,315.752,361.947,170.645,49.274,159.592
C07908=1021.514,316.000,361.913,170.650,49.272,159.592
C07909=1021.521,316.249,361.880,170.656,49.270,159.593
C07910=1021.527,316.496,361.846,170.662,49.267,159.593
C07911=1021.534,316.743,361.812,170.668,49.265,159.593
C07912=1021.541,316.991,361.778,170.674,49.263,159.594
C07913=1021.547,317.238,361.744,170.679,49.260,159.594
C07914=1021.555,317.486,361.711,170.685,49.257,159.594
C07915=1021.562,317.734,361.677,170.691,49.256,159.595
C07916=1021.568,317.981,361.643,170.697,49.253,159.595
C07917=1021.575,318.228,361.609,170.702,49.250,159.595
C07918=1021.582,318.476,361.575,170.709,49.248,159.596
C07919=1021.589,318.724,361.541,170.714,49.246,159.596
C07920=1021.596,318.972,361.507,170.720,49.244,159.597
C07921=1021.602,319.219,361.473,170.726,49.241,159.597
C07922=1021.610,319.466,361.440,170.732,49.239,159.597
C07923=1021.616,319.714,361.404,170.738,49.237,159.598
C07924=1021.624,319.962,361.371,170.743,49.234,159.598
C07925=1021.631,320.209,361.337,170.749,49.232,159.598
C07926=1021.637,320.457,361.302,170.755,49.230,159.599
C07927=1021.644,320.704,361.269,170.761,49.228,159.599
C07928=1021.651,320.952,361.235,170.767,49.226,159.600
C07929=1021.658,321.199,361.200,170.773,49.223,159.600
C07930=1021.665,321.447,361.166,170.779,49.221,159.600
C07931=1021.672,321.687,361.133,170.784,49.219,159.601
C07932=1021.679,321.926,361.100,170.790,49.217,159.601
C07933=1021.686,322.165,361.068,170.797,49.215,159.602
C07934=1021.692,322.405,361.034,170.802,49.212,159.602
C07935=1021.699,322.645,361.001,170.807,49.211,159.602
C07936=1021.706,322.884,360.968,170.813,49.209,159.603
C07937=1021.713,323.124,360.935,170.819,49.206,159.603
C07938=1021.720,323.363,360.901,170.825,49.204,159.604
C07939=1021.727,323.611,360.867,170.831,49.203,159.604
C07940=1021.734,323.859,360.833,170.837,49.200,159.604
C07941=1021.741,324.106,360.798,170.843,49.198,159.605
C07942=1021.748,324.354,360.765,170.849,49.196,159.605
C07943=1021.756,324.601,360.730,170.856,49.194,159.606
C07944=1021.762,324.849,360.696,170.861,49.191,159.606
C07945=1021.770,325.096,360.661,170.867,49.189,159.607
C07946=1021.777,325.343,360.627,170.873,49.187,159.607
C07947=1021.784,325.591,360.592,170.879,49.186,159.607
C07948=1021.792,325.839,360.558,170.886,49.184,159.608
C07949=1021.799,326.086,360.523,170.891,49.181,159.608
C07950=1021.806,326.333,360.488,170.897,49.179,159.609
C07951=1021.813,326.581,360.454,170.904,49.177,159.609
C07952=1021.821,326.828,360.420,170.910,49.175,159.610
C07953=1021.827,327.076,360.385,170.916,49.173,159.610
C07954=1021.834,327.323,360.350,170.922,49.171,159.611
C07955=1021.841,327.571,360.316,170.928,49.169,159.611
C07956=1021.849,327.819,360.280,170.934,49.167,159.612
C07957=1021.855,328.066,360.245,170.941,49.166,159.612
C07958=1021.862,328.313,360.210,170.947,49.164,159.613
C07959=1021.870,328.560,360.175,170.953,49.162,159.613
C07960=1021.876,328.808,360.140,170.959,49.160,159.614
C07961=1021.883,329.055,360.105,170.965,49.158,159.614
C07962=1021.891,329.303,360.070,170.972,49.156,159.615
C07963=1021.898,329.550,360.035,170.978,49.155,159.615
C07964=1021.905,329.798,360.000,170.984,49.153,159.616
C07965=1021.912,330.045,359.965,170.990,49.151,159.616
C07966=1021.919,330.293,359.929,170.996,49.149,159.617
C07967=1021.926,330.540,359.895,171.003,49.148,159.617
C07968=1021.933,330.787,359.860,171.009,49.146,159.618
C07969=1021.940,331.035,359.825,171.015,49.144,159.618
C07970=1021.948,331.282,359.788,171.022,49.141,159.619
C07971=1021.955,331.529,359.754,171.028,49.140,159.620
C07972=1021.962,331.777,359.719,171.034,49.138,159.620
C07973=1021.969,332.025,359.683,171.040,49.136,159.621
C07974=1021.976,332.272,359.648,171.047,49.135,159.621
C07975=1021.984,332.520,359.612,171.053,49.133,159.622
C07976=1021.991,332.767,359.577,171.059,49.132,159.622
C07977=1021.998,333.014,359.542,171.066,49.130,159.623
C07978=1022.005,333.262,359.507,171.073,49.128,159.624
C07979=1022.013,333.509,359.471,171.079,49.126,159.624
C07980=1022.019,333.756,359.436,171.085,49.125,159.625
C07981=1022.027,334.004,359.399,171.091,49.123,159.625
C07982=1022.034,334.251,359.364,171.097,49.122,159.626
C07983=1022.041,334.498,359.328,171.104,49.120,159.626
C07984=1022.048,334.746,359.293,171.111,49.118,159.627
C07985=1022.056,334.993,359.257,171.117,49.117,159.628
C07986=1022.063,335.241,359.222,171.123,49.115,159.628
C07987=1022.070,335.487,359.186,171.130,49.114,159.629
C07988=1022.077,335.735,359.150,171.136,49.112,159.629
C07989=1022.084,335.982,359.114,171.143,49.110,159.630
C07990=1022.092,336.230,359.078,171.149,49.109,159.631
C07991=1022.099,336.467,359.044,171.156,49.108,159.631
C07992=1022.105,336.705,359.010,171.162,49.106,159.632
C07993=1022.112,336.942,358.975,171.168,49.104,159.632
C07994=1022.120,337.179,358.941,171.175,49.103,159.633
C07995=1022.127,337.417,358.906,171.181,49.102,159.634
C07996=1022.134,337.653,358.872,171.187,49.100,159.634
C07997=1022.140,337.891,358.837,171.193,49.099,159.635
C07998=1022.148,338.128,358.803,171.200,49.097,159.636
C07999=1022.155,338.375,358.767,171.206,49.096,159.636
C08000=1022.162,338.623,358.731,171.213,49.095,159.637
C08001=1022.170,338.871,358.695,171.219,49.093,159.638
C08002=1022.177,339.117,358.659,171.226,49.091,159.638
C08003=1022.185,339.365,358.623,171.232,49.090,159.639
C08004=1022.192,339.612,358.587,171.239,49.088,159.639
C08005=1022.199,339.859,358.551,171.245,49.087,159.640
C08006=1022.206,340.107,358.514,171.252,49.086,159.641
C08007=1022.214,340.354,358.478,171.259,49.084,159.642
C08008=1022.221,340.601,358.442,171.266,49.084,159.642
C08009=1022.229,340.848,358.406,171.272,49.082,159.643
C08010=1022.236,341.096,358.369,171.279,49.081,159.644
C08011=1022.244,341.343,358.332,171.286,49.079,159.644
C08012=1022.251,341.590,358.296,171.292,49.078,159.645
C08013=1022.258,341.837,358.260,171.299,49.077,159.646
C08014=1022.265,342.085,358.223,171.306,49.075,159.647
C08015=1022.273,342.332,358.187,171.313,49.074,159.647
C08016=1022.280,342.578,358.150,171.319,49.073,159.648
C08017=1022.287,342.826,358.114,171.326,49.072,159.649
C08018=1022.295,343.074,358.077,171.333,49.070,159.649
C08019=1022.303,343.320,358.040,171.340,49.070,159.650
C08020=1022.310,343.568,358.004,171.347,49.068,159.651
C08021=1022.317,343.815,357.968,171.353,49.067,159.652
C08022=1022.325,344.062,357.931,171.360,49.066,159.653
C08023=1022.332,344.310,357.894,171.367,49.064,159.653
C08024=1022.340,344.556,357.857,171.374,49.063,159.654
C08025=1022.348,344.804,357.821,171.381,49.062,159.655
C08026=1022.355,345.051,357.783,171.388,49.061,159.656
C08027=1022.363,345.298,357.747,171.395,49.060,159.656
C08028=1022.370,345.545,357.710,171.401,49.059,159.657
C08029=1022.378,345.793,357.673,171.408,49.057,159.658
C08030=1022.385,346.040,357.636,171.415,49.056,159.659
C08031=1022.393,346.287,357.599,171.422,49.055,159.659
C08032=1022.400,346.534,357.563,171.429,49.054,159.660
C08033=1022.408,346.781,357.526,171.436,49.053,159.661
C08034=1022.416,347.028,357.488,171.443,49.052,159.662
C08035=1022.423,347.276,357.452,171.450,49.051,159.663
C08036=1022.431,347.523,357.414,171.456,49.050,159.663
C08037=1022.439,347.770,357.378,171.464,49.049,159.664
C08038=1022.446,348.017,357.340,171.471,49.048,159.665
C08039=1022.454,348.264,357.303,171.477,49.047,159.666
C08040=1022.461,348.511,357.266,171.485,49.046,159.667
C08041=1022.469,348.758,357.229,171.492,49.045,159.668
C08042=1022.476,349.005,357.192,171.500,49.044,159.669
C08043=1022.483,349.253,357.154,171.506,49.043,159.669
C08044=1022.491,349.499,357.117,171.514,49.042,159.670
C08045=1022.498,349.746,357.080,171.520,49.041,159.671
C08046=1022.506,349.994,357.042,171.527,49.040,159.672
C08047=1022.514,350.241,357.005,171.535,49.039,159.673
C08048=1022.521,350.488,356.967,171.542,49.039,159.674
C08049=1022.529,350.735,356.929,171.549,49.038,159.675
C08050=1022.537,350.982,356.892,171.556,49.036,159.675
C08051=1022.545,351.218,356.856,171.562,49.036,159.676
C08052=1022.552,351.453,356.820,171.569,49.035,159.677
C08053=1022.559,351.689,356.785,171.577,49.034,159.678
C08054=1022.567,351.926,356.750,171.584,49.033,159.679
C08055=1022.573,352.161,356.713,171.590,49.033,159.680
C08056=1022.581,352.396,356.677,171.597,49.032,159.681
C08057=1022.589,352.632,356.641,171.604,49.031,159.681
C08058=1022.596,352.868,356.605,171.612,49.030,159.682
C08059=1022.604,353.115,356.568,171.618,49.030,159.683
C08060=1022.612,353.362,356.530,171.626,49.029,159.684
C08061=1022.619,353.609,356.492,171.633,49.028,159.685
C08062=1022.628,353.857,356.455,171.641,49.027,159.686
C08063=1022.635,354.103,356.416,171.647,49.026,159.687
C08064=1022.642,354.350,356.379,171.655,49.026,159.688
C08065=1022.651,354.597,356.341,171.662,49.025,159.689
C08066=1022.659,354.844,356.303,171.670,49.024,159.690
C08067=1022.666,355.091,356.265,171.677,49.024,159.691
C08068=1022.674,355.339,356.227,171.685,49.023,159.692
C08069=1022.682,355.585,356.189,171.692,49.022,159.693
C08070=1022.690,355.832,356.150,171.699,49.022,159.694
C08071=1022.698,356.079,356.113,171.707,49.021,159.695
C08072=1022.706,356.326,356.075,171.714,49.020,159.695
C08073=1022.713,356.573,356.037,171.722,49.020,159.697
C08074=1022.722,356.820,355.998,171.729,49.019,159.697
C08075=1022.729,357.067,355.960,171.737,49.019,159.699
C08076=1022.737,357.314,355.922,171.745,49.018,159.699
C08077=1022.744,357.561,355.884,171.752,49.018,159.701
C08078=1022.753,357.808,355.846,171.759,49.017,159.701
C08079=1022.761,358.054,355.807,171.766,49.017,159.703
C08080=1022.769,358.302,355.769,171.774,49.016,159.703
C08081=1022.777,358.548,355.731,171.782,49.015,159.705
C08082=1022.785,358.795,355.692,171.789,49.015,159.706
C08083=1022.793,359.042,355.653,171.797,49.014,159.707
C08084=1022.800,359.289,355.615,171.805,49.014,159.708
C08085=1022.809,359.536,355.576,171.812,49.014,159.709
C08086=1022.817,359.783,355.538,171.820,49.013,159.710
C08087=1022.824,360.030,355.500,171.828,49.012,159.711
C08088=1022.832,360.277,355.461,171.835,49.012,159.712
C08089=1022.840,360.524,355.423,171.843,49.012,159.713
C08090=1022.848,360.770,355.383,171.851,49.011,159.714
C08091=1022.857,361.017,355.345,171.858,49.011,159.715
C08092=1022.863,361.264,355.306,171.866,49.010,159.716
C08093=1022.872,361.511,355.267,171.874,49.010,159.717
C08094=1022.880,361.758,355.228,171.881,49.010,159.718
C08095=1022.888,362.005,355.189,171.889,49.009,159.719
C08096=1022.896,362.251,355.150,171.898,49.009,159.721
C08097=1022.904,362.498,355.112,171.905,49.009,159.722
C08098=1022.912,362.745,355.072,171.913,49.008,159.723
C08099=1022.920,362.993,355.033,171.921,49.008,159.724
C08100=1022.929,363.239,354.994,171.929,49.008,159.725
C08101=1022.936,363.486,354.956,171.936,49.007,159.726
C08102=1022.945,363.732,354.916,171.944,49.008,159.727
C08103=1022.953,363.979,354.877,171.953,49.007,159.729
C08104=1022.960,364.226,354.838,171.961,49.007,159.730
C08105=1022.969,364.473,354.799,171.968,49.007,159.731
C08106=1022.977,364.720,354.759,171.976,49.006,159.732
C08107=1022.985,364.967,354.721,171.984,49.006,159.733
C08108=1022.994,365.213,354.681,171.992,49.006,159.734
C08109=1023.002,365.460,354.641,172.000,49.006,159.735
C08110=1023.010,365.706,354.602,172.008,49.005,159.737
C08111=1023.018,365.946,354.565,172.016,49.005,159.738
C08112=1023.026,366.185,354.526,172.024,49.005,159.739
C08113=1023.034,366.425,354.488,172.031,49.005,159.740
C08114=1023.042,366.664,354.450,172.039,49.005,159.741
C08115=1023.050,366.903,354.412,172.047,49.004,159.742
C08116=1023.059,367.142,354.374,172.055,49.005,159.744
C08117=1023.066,367.381,354.336,172.063,49.004,159.745
C08118=1023.074,367.620,354.297,172.071,49.004,159.746
C08119=1023.083,367.867,354.258,172.079,49.004,159.747
C08120=1023.091,368.114,354.219,172.087,49.004,159.748
C08121=1023.099,368.360,354.179,172.096,49.004,159.750
C08122=1023.107,368.607,354.140,172.103,49.005,159.751
C08123=1023.116,368.854,354.099,172.111,49.004,159.752
C08124=1023.124,369.101,354.059,172.120,49.004,159.753
C08125=1023.132,369.348,354.019,172.128,49.004,159.755
C08126=1023.141,369.593,353.979,172.136,49.004,159.756
C08127=1023.149,369.840,353.939,172.145,49.004,159.757
C08128=1023.157,370.087,353.900,172.153,49.004,159.758
C08129=1023.165,370.333,353.859,172.162,49.005,159.760
C08130=1023.174,370.581,353.820,172.170,49.005,159.761
C08131=1023.182,370.827,353.779,172.179,49.005,159.762
C08132=1023.191,371.073,353.740,172.187,49.005,159.764
C08133=1023.199,371.320,353.699,172.195,49.005,159.765
C08134=1023.208,371.567,353.659,172.204,49.005,159.766
C08135=1023.216,371.813,353.619,172.212,49.005,159.768
C08136=1023.224,372.060,353.579,172.220,49.005,159.769
C08137=1023.233,372.307,353.538,172.229,49.005,159.770
C08138=1023.242,372.553,353.498,172.237,49.006,159.772
C08139=1023.249,372.800,353.459,172.246,49.006,159.773
C08140=1023.259,373.046,353.418,172.254,49.006,159.774
C08141=1023.267,373.293,353.377,172.263,49.006,159.776
C08142=1023.275,373.539,353.337,172.271,49.006,159.777
C08143=1023.284,373.786,353.297,172.280,49.007,159.778
C08144=1023.292,374.033,353.257,172.288,49.007,159.780
C08145=1023.301,374.279,353.216,172.297,49.007,159.781
C08146=1023.309,374.526,353.175,172.305,49.008,159.782
C08147=1023.319,374.772,353.135,172.314,49.008,159.784
C08148=1023.327,375.019,353.094,172.323,49.008,159.785
C08149=1023.336,375.265,353.054,172.332,49.008,159.787
C08150=1023.344,375.511,353.013,172.340,49.008,159.788
C08151=1023.353,375.758,352.973,172.349,49.009,159.790
C08152=1023.361,376.004,352.932,172.358,49.009,159.791
C08153=1023.371,376.251,352.892,172.366,49.010,159.792
C08154=1023.379,376.498,352.851,172.376,49.010,159.794
C08155=1023.387,376.744,352.810,172.384,49.010,159.795
C08156=1023.397,376.990,352.769,172.393,49.011,159.797
C08157=1023.405,377.237,352.729,172.401,49.011,159.798
C08158=1023.414,377.484,352.688,172.410,49.012,159.800
C08159=1023.423,377.730,352.646,172.419,49.013,159.801
C08160=1023.431,377.976,352.605,172.429,49.012,159.802
C08161=1023.440,378.223,352.563,172.437,49.013,159.804
C08162=1023.448,378.470,352.522,172.446,49.014,159.806
C08163=1023.457,378.715,352.481,172.455,49.014,159.807
C08164=1023.466,378.962,352.441,172.464,49.014,159.808
C08165=1023.475,379.208,352.399,172.473,49.015,159.810
C08166=1023.483,379.455,352.358,172.482,49.016,159.812
C08167=1023.492,379.701,352.317,172.490,49.016,159.813
C08168=1023.501,379.947,352.275,172.500,49.017,159.814
C08169=1023.509,380.194,352.234,172.509,49.017,159.816
C08170=1023.518,380.441,352.192,172.518,49.018,159.818
C08171=1023.528,380.694,352.150,172.528,49.018,159.819
C08172=1023.537,380.948,352.108,172.536,49.019,159.821
C08173=1023.545,381.201,352.064,172.546,49.020,159.822
C08174=1023.555,381.454,352.022,172.555,49.021,159.824
C08175=1023.564,381.701,351.980,172.565,49.021,159.826
C08176=1023.573,381.947,351.939,172.574,49.022,159.827
C08177=1023.582,382.194,351.897,172.584,49.023,159.829
C08178=1023.591,382.441,351.856,172.593,49.023,159.830
C08179=1023.600,382.687,351.814,172.601,49.024,159.832
C08180=1023.608,382.932,351.772,172.611,49.024,159.833
C08181=1023.618,383.179,351.730,172.620,49.025,159.835
C08182=1023.627,383.425,351.689,172.630,49.026,159.837
C08183=1023.636,383.671,351.647,172.639,49.027,159.838
C08184=1023.645,383.918,351.606,172.649,49.027,159.840
C08185=1023.654,384.164,351.564,172.658,49.029,159.842
C08186=1023.663,384.411,351.522,172.668,49.029,159.843
C08187=1023.672,384.657,351.480,172.677,49.030,159.845
C08188=1023.681,384.903,351.438,172.687,49.031,159.847
C08189=1023.690,385.149,351.396,172.695,49.032,159.848
C08190=1023.700,385.395,351.355,172.706,49.033,159.850
C08191=1023.710,385.642,351.312,172.714,49.033,159.852
C08192=1023.719,385.888,351.271,172.725,49.034,159.853
C08193=1023.728,386.134,351.228,172.733,49.035,159.855
C08194=1023.736,386.380,351.186,172.744,49.036,159.857
C08195=1023.745,386.626,351.143,172.753,49.036,159.858
C08196=1023.755,386.873,351.101,172.763,49.038,159.860
C08197=1023.764,387.119,351.059,172.773,49.039,159.862
C08198=1023.773,387.365,351.016,172.782,49.040,159.864
C08199=1023.782,387.611,350.975,172.792,49.040,159.865
C08200=1023.792,387.857,350.932,172.802,49.041,159.867
C08201=1023.801,388.103,350.890,172.811,49.043,159.869
C08202=1023.810,388.349,350.846,172.821,49.044,159.871
C08203=1023.820,388.596,350.804,172.831,49.045,159.872
C08204=1023.829,388.842,350.762,172.840,49.046,159.874
C08205=1023.839,389.088,350.719,172.851,49.047,159.876
C08206=1023.848,389.334,350.677,172.861,49.048,159.878
C08207=1023.856,389.580,350.634,172.870,49.049,159.880
C08208=1023.866,389.827,350.591,172.880,49.050,159.881
C08209=1023.876,390.072,350.548,172.890,49.051,159.883
C08210=1023.885,390.319,350.504,172.899,49.052,159.885
C08211=1023.894,390.564,350.462,172.910,49.053,159.887
C08212=1023.904,390.811,350.419,172.920,49.054,159.889
C08213=1023.912,391.057,350.376,172.930,49.056,159.891
C08214=1023.922,391.303,350.333,172.940,49.057,159.892
C08215=1023.932,391.548,350.290,172.950,49.058,159.894
C08216=1023.942,391.795,350.247,172.960,49.060,159.896
C08217=1023.950,392.041,350.204,172.970,49.061,159.898
C08218=1023.960,392.287,350.161,172.980,49.062,159.900
C08219=1023.970,392.533,350.118,172.991,49.063,159.902
C08220=1023.979,392.779,350.074,173.001,49.064,159.904
C08221=1023.989,393.025,350.031,173.011,49.066,159.906
C08222=1023.999,393.271,349.988,173.021,49.067,159.907
C08223=1024.007,393.517,349.945,173.031,49.068,159.909
C08224=1024.018,393.763,349.901,173.041,49.069,159.911
C08225=1024.027,394.009,349.857,173.052,49.071,159.913
C08226=1024.037,394.255,349.814,173.063,49.072,159.915
C08227=1024.046,394.501,349.771,173.073,49.073,159.917
C08228=1024.056,394.747,349.727,173.083,49.075,159.919
C08229=1024.065,394.993,349.683,173.094,49.076,159.921
C08230=1024.075,395.239,349.640,173.104,49.078,159.923
C08231=1024.086,395.529,349.588,173.116,49.080,159.926
C08232=1024.098,395.820,349.537,173.129,49.081,159.928
C08233=1024.109,396.109,349.485,173.141,49.083,159.930
C08234=1024.120,396.399,349.433,173.154,49.085,159.933
C08235=1024.131,396.645,349.390,173.164,49.086,159.935
C08236=1024.140,396.891,349.346,173.175,49.088,159.937
C08237=1024.150,397.137,349.302,173.185,49.089,159.939
C08238=1024.160,397.383,349.257,173.196,49.091,159.941
C08239=1024.170,397.629,349.214,173.207,49.093,159.943
C08240=1024.179,397.875,349.170,173.217,49.094,159.945
C08241=1024.189,398.121,349.126,173.228,49.096,159.947
C08242=1024.200,398.367,349.081,173.239,49.097,159.949
C08243=1024.209,398.613,349.037,173.250,49.098,159.951
C08244=1024.220,398.858,348.993,173.261,49.100,159.953
C08245=1024.229,399.104,348.949,173.271,49.102,159.955
C08246=1024.239,399.350,348.904,173.282,49.104,159.958
C08247=1024.249,399.596,348.860,173.294,49.105,159.960
C08248=1024.259,399.841,348.815,173.304,49.107,159.962
C08249=1024.268,400.087,348.771,173.315,49.109,159.964
C08250=1024.279,400.333,348.727,173.326,49.110,159.966
C08251=1024.289,400.579,348.682,173.338,49.112,159.968
C08252=1024.299,400.824,348.637,173.348,49.114,159.971
C08253=1024.308,401.070,348.593,173.359,49.116,159.973
C08254=1024.319,401.316,348.548,173.371,49.117,159.975
C08255=1024.329,401.562,348.504,173.382,49.119,159.977
C08256=1024.338,401.807,348.459,173.393,49.121,159.979
C08257=1024.349,402.053,348.413,173.404,49.123,159.981
C08258=1024.358,402.299,348.369,173.415,49.125,159.984
C08259=1024.368,402.544,348.324,173.426,49.127,159.986
C08260=1024.379,402.790,348.278,173.438,49.128,159.988
C08261=1024.389,403.036,348.233,173.449,49.131,159.990
C08262=1024.400,403.281,348.189,173.460,49.133,159.993
C08263=1024.409,403.527,348.144,173.472,49.134,159.995
C08264=1024.419,403.772,348.098,173.483,49.136,159.997
C08265=1024.430,404.018,348.053,173.494,49.138,160.000
C08266=1024.439,404.264,348.008,173.505,49.140,160.002
C08267=1024.450,404.509,347.962,173.518,49.142,160.004
C08268=1024.460,404.755,347.917,173.528,49.144,160.007
C08269=1024.470,405.001,347.872,173.540,49.146,160.009
C08270=1024.481,405.247,347.826,173.552,49.148,160.011
C08271=1024.491,405.491,347.781,173.564,49.150,160.014
C08272=1024.502,405.737,347.736,173.575,49.152,160.016
C08273=1024.512,405.983,347.690,173.586,49.154,160.018
C08274=1024.523,406.229,347.645,173.599,49.156,160.021
C08275=1024.533,406.474,347.600,173.610,49.158,160.023
C08276=1024.543,406.720,347.554,173.622,49.161,160.026
C08277=1024.554,406.965,347.508,173.634,49.162,160.028
C08278=1024.564,407.211,347.463,173.646,49.165,160.030
C08279=1024.575,407.457,347.417,173.657,49.167,160.033
C08280=1024.585,407.702,347.371,173.669,49.169,160.035
C08281=1024.595,407.948,347.325,173.681,49.171,160.038
C08282=1024.606,408.193,347.279,173.694,49.174,160.040
C08283=1024.617,408.438,347.234,173.706,49.176,160.043
C08284=1024.628,408.684,347.188,173.717,49.178,160.045
C08285=1024.639,408.930,347.142,173.729,49.180,160.047
C08286=1024.649,409.175,347.096,173.741,49.182,160.050
C08287=1024.660,409.421,347.050,173.754,49.185,160.053
C08288=1024.671,409.666,347.004,173.766,49.187,160.055
C08289=1024.682,409.911,346.958,173.778,49.189,160.058
C08290=1024.691,410.157,346.911,173.790,49.191,160.060
C08291=1024.705,410.471,346.852,173.806,49.195,160.063
C08292=1024.719,410.782,346.793,173.821,49.198,160.067
C08293=1024.733,411.096,346.734,173.837,49.201,160.070
C08294=1024.746,411.408,346.675,173.852,49.204,160.073
C08295=1024.757,411.654,346.627,173.865,49.206,160.076
C08296=1024.768,411.899,346.581,173.877,49.209,160.078
C08297=1024.779,412.145,346.535,173.890,49.211,160.081
C08298=1024.790,412.390,346.488,173.902,49.214,160.084
C08299=1024.801,412.635,346.441,173.915,49.216,160.086
C08300=1024.811,412.881,346.394,173.927,49.219,160.089
C08301=1024.822,413.126,346.347,173.941,49.221,160.092
C08302=1024.834,413.371,346.300,173.953,49.224,160.095
C08303=1024.845,413.616,346.254,173.966,49.226,160.097
C08304=1024.855,413.862,346.207,173.978,49.229,160.100
C08305=1024.866,414.107,346.160,173.991,49.231,160.103
C08306=1024.877,414.352,346.113,174.005,49.234,160.105
C08307=1024.889,414.598,346.066,174.017,49.237,160.108
C08308=1024.899,414.843,346.019,174.030,49.239,160.111
C08309=1024.911,415.089,345.972,174.042,49.242,160.113
C08310=1024.922,415.334,345.924,174.056,49.244,160.116
C08311=1024.933,415.579,345.877,174.069,49.247,160.119
C08312=1024.944,415.825,345.830,174.081,49.250,160.122
C08313=1024.956,416.070,345.782,174.095,49.252,160.125
C08314=1024.966,416.315,345.735,174.108,49.255,160.127
C08315=1024.978,416.560,345.687,174.120,49.258,160.130
C08316=1024.989,416.806,345.640,174.134,49.261,160.133
C08317=1025.000,417.051,345.592,174.147,49.264,160.136
C08318=1025.011,417.296,345.544,174.161,49.266,160.139
C08319=1025.023,417.541,345.496,174.174,49.269,160.142
C08320=1025.033,417.786,345.449,174.187,49.272,160.145
C08321=1025.045,418.031,345.401,174.200,49.275,160.148
C08322=1025.056,418.277,345.353,174.214,49.278,160.151
C08323=1025.068,418.522,345.305,174.227,49.281,160.153
C08324=1025.079,418.767,345.257,174.241,49.284,160.156
C08325=1025.091,419.012,345.209,174.255,49.286,160.159
C08326=1025.102,419.258,345.161,174.268,49.289,160.162
C08327=1025.114,419.503,345.113,174.282,49.292,160.165
C08328=1025.125,419.748,345.065,174.296,49.295,160.168
C08329=1025.137,419.992,345.017,174.309,49.298,160.171
C08330=1025.148,420.238,344.968,174.323,49.301,160.174
C08331=1025.160,420.483,344.921,174.337,49.304,160.177
C08332=1025.171,420.728,344.872,174.351,49.307,160.180
C08333=1025.183,420.973,344.824,174.364,49.310,160.183
C08334=1025.194,421.218,344.776,174.378,49.313,160.186
C08335=1025.207,421.462,344.727,174.392,49.317,160.190
C08336=1025.218,421.709,344.679,174.406,49.320,160.193
C08337=1025.230,421.953,344.630,174.420,49.322,160.196
C08338=1025.242,422.198,344.581,174.435,49.326,160.199
C08339=1025.253,422.444,344.532,174.449,49.329,160.202
C08340=1025.265,422.689,344.483,174.463,49.332,160.205
C08341=1025.277,422.933,344.435,174.477,49.335,160.208
C08342=1025.288,423.178,344.386,174.492,49.339,160.212
C08343=1025.300,423.423,344.337,174.506,49.341,160.215
C08344=1025.313,423.668,344.288,174.520,49.345,160.218
C08345=1025.325,423.913,344.239,174.534,49.348,160.221
C08346=1025.336,424.158,344.190,174.548,49.351,160.224
C08347=1025.347,424.402,344.141,174.563,49.354,160.227
C08348=1025.360,424.648,344.092,174.577,49.358,160.231
C08349=1025.372,424.892,344.042,174.592,49.361,160.234
C08350=1025.384,425.137,343.993,174.607,49.364,160.237
C08351=1025.398,425.404,343.939,174.623,49.368,160.241
C08352=1025.411,425.672,343.885,174.639,49.372,160.245
C08353=1025.423,425.938,343.831,174.655,49.376,160.248
C08354=1025.437,426.205,343.778,174.670,49.379,160.252
C08355=1025.449,426.451,343.728,174.686,49.382,160.255
C08356=1025.461,426.696,343.678,174.701,49.386,160.258
C08357=1025.473,426.940,343.629,174.715,49.390,160.262
C08358=1025.485,427.185,343.578,174.731,49.393,160.265
C08359=1025.498,427.429,343.528,174.745,49.397,160.268
C08360=1025.510,427.675,343.479,174.761,49.400,160.272
C08361=1025.521,427.919,343.429,174.776,49.404,160.276
C08362=1025.534,428.164,343.379,174.791,49.407,160.279
C08363=1025.549,428.465,343.317,174.810,49.412,160.283
C08364=1025.564,428.766,343.256,174.829,49.416,160.288
C08365=1025.580,429.068,343.193,174.848,49.421,160.292
C08366=1025.595,429.368,343.132,174.867,49.425,160.296
C08367=1025.608,429.613,343.082,174.883,49.429,160.300
C08368=1025.620,429.858,343.032,174.897,49.433,160.303
C08369=1025.632,430.102,342.981,174.913,49.436,160.307
C08370=1025.645,430.347,342.931,174.929,49.440,160.310
C08371=1025.657,430.591,342.880,174.945,49.443,160.314
C08372=1025.670,430.836,342.830,174.959,49.447,160.317
C08373=1025.682,431.080,342.779,174.976,49.451,160.321
C08374=1025.696,431.325,342.728,174.991,49.455,160.325
C08375=1025.708,431.570,342.678,175.008,49.459,160.328
C08376=1025.720,431.814,342.627,175.023,49.462,160.332
C08377=1025.734,432.059,342.576,175.040,49.466,160.336
C08378=1025.746,432.303,342.525,175.055,49.470,160.339
C08379=1025.759,432.548,342.475,175.071,49.474,160.343
C08380=1025.772,432.793,342.424,175.088,49.478,160.347
C08381=1025.784,433.037,342.373,175.104,49.482,160.351
C08382=1025.798,433.282,342.321,175.120,49.486,160.354
C08383=1025.811,433.526,342.270,175.137,49.490,160.358
C08384=1025.824,433.771,342.219,175.153,49.494,160.362
C08385=1025.836,434.015,342.168,175.170,49.498,160.366
C08386=1025.850,434.259,342.116,175.186,49.502,160.370
C08387=1025.863,434.503,342.065,175.203,49.505,160.373
C08388=1025.875,434.748,342.013,175.219,49.509,160.377
C08389=1025.889,434.993,341.962,175.236,49.514,160.381
C08390=1025.902,435.237,341.910,175.253,49.517,160.385
C08391=1025.915,435.481,341.859,175.269,49.522,160.389
C08392=1025.928,435.726,341.807,175.285,49.526,160.393
C08393=1025.941,435.970,341.755,175.303,49.530,160.397
C08394=1025.954,436.214,341.703,175.320,49.535,160.401
C08395=1025.968,436.458,341.651,175.337,49.538,160.405
C08396=1025.981,436.702,341.599,175.353,49.543,160.409
C08397=1025.995,436.947,341.547,175.371,49.547,160.413
C08398=1026.007,437.191,341.495,175.388,49.551,160.417
C08399=1026.021,437.435,341.443,175.405,49.555,160.421
C08400=1026.034,437.680,341.391,175.423,49.560,160.425
C08401=1026.048,437.923,341.339,175.440,49.564,160.429
C08402=1026.061,438.168,341.286,175.458,49.568,160.433
C08403=1026.075,438.412,341.234,175.474,49.572,160.437
C08404=1026.088,438.656,341.182,175.492,49.577,160.441
C08405=1026.101,438.901,341.129,175.510,49.581,160.446
C08406=1026.115,439.144,341.077,175.528,49.586,160.450
C08407=1026.129,439.388,341.024,175.545,49.590,160.454
C08408=1026.142,439.633,340.971,175.563,49.594,160.458
C08409=1026.156,439.877,340.918,175.581,49.598,160.462
C08410=1026.170,440.120,340.866,175.599,49.603,160.467
C08411=1026.182,440.340,340.818,175.615,49.607,160.470
C08412=1026.194,440.560,340.771,175.631,49.611,160.474
C08413=1026.207,440.780,340.723,175.648,49.615,160.478
C08414=1026.220,440.999,340.676,175.664,49.619,160.482
C08415=1026.232,441.218,340.627,175.680,49.623,160.486
C08416=1026.245,441.438,340.579,175.697,49.627,160.490
C08417=1026.257,441.658,340.532,175.713,49.631,160.494
C08418=1026.270,441.877,340.484,175.729,49.635,160.498
C08419=1026.284,442.120,340.431,175.748,49.640,160.502
C08420=1026.298,442.363,340.378,175.766,49.645,160.506
C08421=1026.313,442.607,340.324,175.785,49.649,160.511
C08422=1026.326,442.851,340.272,175.803,49.654,160.515
C08423=1026.341,443.094,340.220,175.822,49.658,160.520
C08424=1026.357,443.337,340.167,175.841,49.662,160.524
C08425=1026.373,443.581,340.115,175.859,49.667,160.528
C08426=1026.389,443.825,340.065,175.878,49.671,160.533
C08427=1026.406,444.068,340.014,175.897,49.675,160.537
C08428=1026.423,444.312,339.964,175.917,49.679,160.542
C08429=1026.442,444.556,339.913,175.936,49.683,160.546
C08430=1026.460,444.800,339.863,175.955,49.687,160.550
C08431=1026.478,445.044,339.815,175.975,49.691,160.555
C08432=1026.497,445.288,339.766,175.994,49.695,160.559
C08433=1026.517,445.532,339.717,176.013,49.699,160.563
C08434=1026.537,445.776,339.669,176.033,49.702,160.568
C08435=1026.557,446.021,339.621,176.053,49.706,160.572
C08436=1026.578,446.265,339.574,176.073,49.709,160.576
C08437=1026.600,446.510,339.527,176.093,49.713,160.581
C08438=1026.621,446.754,339.481,176.112,49.716,160.585
C08439=1026.644,446.998,339.434,176.132,49.720,160.589
C08440=1026.667,447.243,339.389,176.153,49.723,160.594
C08441=1026.690,447.488,339.344,176.173,49.726,160.598
C08442=1026.714,447.733,339.298,176.193,49.729,160.602
C08443=1026.738,447.978,339.254,176.213,49.733,160.607
C08444=1026.763,448.223,339.210,176.234,49.736,160.611
C08445=1026.787,448.467,339.166,176.254,49.738,160.615
C08446=1026.813,448.713,339.123,176.275,49.742,160.620
C08447=1026.839,448.958,339.080,176.295,49.744,160.624
C08448=1026.866,449.203,339.037,176.316,49.747,160.628
C08449=1026.893,449.448,338.995,176.338,49.750,160.633
C08450=1026.920,449.693,338.953,176.358,49.753,160.637
C08451=1026.948,449.938,338.913,176.380,49.755,160.641
C08452=1026.976,450.184,338.871,176.400,49.758,160.645
C08453=1027.004,450.430,338.830,176.422,49.760,160.650
C08454=1027.034,450.675,338.790,176.443,49.762,160.654
C08455=1027.064,450.920,338.750,176.465,49.765,160.658
C08456=1027.093,451.166,338.711,176.486,49.767,160.663
C08457=1027.124,451.411,338.671,176.508,49.769,160.667
C08458=1027.156,451.656,338.633,176.530,49.772,160.671
C08459=1027.187,451.902,338.595,176.552,49.774,160.676
C08460=1027.219,452.148,338.557,176.573,49.776,160.680
C08461=1027.251,452.394,338.519,176.595,49.778,160.684
C08462=1027.284,452.638,338.482,176.618,49.780,160.688
C08463=1027.317,452.885,338.445,176.639,49.782,160.693
C08464=1027.351,453.131,338.409,176.662,49.784,160.697
C08465=1027.385,453.376,338.373,176.684,49.786,160.701
C08466=1027.420,453.622,338.338,176.707,49.788,160.706
C08467=1027.456,453.868,338.303,176.730,49.789,160.710
C08468=1027.491,454.114,338.268,176.752,49.791,160.714
C08469=1027.528,454.359,338.234,176.775,49.792,160.718
C08470=1027.564,454.605,338.200,176.798,49.794,160.723
C08471=1027.290,454.683,337.861,176.801,49.854,160.742
C08472=1027.254,454.438,337.896,176.778,49.853,160.738
C08473=1027.218,454.192,337.930,176.755,49.850,160.733
C08474=1027.181,453.946,337.965,176.732,49.849,160.729
C08475=1027.146,453.700,337.999,176.709,49.847,160.725
C08476=1027.112,453.455,338.035,176.687,49.846,160.721
C08477=1027.077,453.209,338.070,176.665,49.844,160.717
C08478=1027.043,452.963,338.107,176.642,49.842,160.712
C08479=1027.010,452.717,338.143,176.620,49.840,160.708
C08480=1026.977,452.472,338.180,176.597,49.839,160.704
C08481=1026.944,452.226,338.217,176.575,49.837,160.699
C08482=1026.911,451.980,338.255,176.554,49.835,160.695
C08483=1026.880,451.735,338.293,176.531,49.833,160.691
C08484=1026.849,451.489,338.332,176.510,49.831,160.687
C08485=1026.818,451.243,338.371,176.487,49.829,160.682
C08486=1026.788,450.998,338.410,176.466,49.826,160.678
C08487=1026.757,450.752,338.450,176.445,49.824,160.674
C08488=1026.729,450.507,338.490,176.423,49.822,160.669
C08489=1026.700,450.262,338.530,176.401,49.819,160.665
C08490=1026.671,450.016,338.571,176.381,49.817,160.661
C08491=1026.643,449.771,338.612,176.360,49.815,160.657
C08492=1026.615,449.525,338.654,176.338,49.812,160.652
C08493=1026.588,449.281,338.696,176.317,49.809,160.648
C08494=1026.561,449.036,338.739,176.297,49.807,160.644
C08495=1026.536,448.790,338.781,176.275,49.804,160.639
C08496=1026.510,448.545,338.824,176.255,49.801,160.635
C08497=1026.484,448.300,338.868,176.234,49.798,160.631
C08498=1026.460,448.056,338.911,176.213,49.796,160.626
C08499=1026.435,447.811,338.956,176.193,49.792,160.622
C08500=1026.411,447.566,339.000,176.173,49.789,160.618
C08501=1026.388,447.321,339.046,176.152,49.786,160.613
C08502=1026.365,447.076,339.092,176.133,49.783,160.609
C08503=1026.343,446.832,339.138,176.112,49.780,160.605
C08504=1026.321,446.587,339.184,176.092,49.777,160.601
C08505=1026.299,446.343,339.231,176.072,49.773,160.596
C08506=1026.278,446.099,339.278,176.053,49.770,160.592
C08507=1026.257,445.854,339.326,176.033,49.766,160.588
C08508=1026.236,445.609,339.373,176.013,49.763,160.583
C08509=1026.218,445.365,339.421,175.993,49.759,160.579
C08510=1026.198,445.122,339.470,175.973,49.755,160.574
C08511=1026.178,444.878,339.519,175.955,49.752,160.570
C08512=1026.160,444.633,339.568,175.935,49.748,160.566
C08513=1026.143,444.389,339.618,175.916,49.744,160.562
C08514=1026.125,444.145,339.669,175.897,49.740,160.557
C08515=1026.108,443.902,339.719,175.878,49.736,160.553
C08516=1026.092,443.658,339.770,175.858,49.732,160.548
C08517=1026.076,443.415,339.822,175.840,49.728,160.544
C08518=1026.060,443.171,339.873,175.821,49.724,160.540
C08519=1026.044,442.928,339.925,175.802,49.720,160.535
C08520=1026.029,442.684,339.978,175.783,49.715,160.531
C08521=1026.015,442.441,340.030,175.765,49.710,160.526
C08522=1026.001,442.198,340.084,175.746,49.706,160.522
C08523=1025.987,441.955,340.137,175.728,49.702,160.518
C08524=1025.975,441.739,340.184,175.712,49.698,160.514
C08525=1025.962,441.524,340.230,175.695,49.694,160.510
C08526=1025.950,441.308,340.277,175.679,49.690,160.506
C08527=1025.937,441.092,340.324,175.663,49.686,160.502
C08528=1025.925,440.877,340.372,175.648,49.682,160.499
C08529=1025.913,440.662,340.418,175.631,49.678,160.495
C08530=1025.901,440.446,340.465,175.615,49.674,160.491
C08531=1025.888,440.231,340.511,175.599,49.670,160.487
C08532=1025.875,439.987,340.564,175.581,49.666,160.483
C08533=1025.861,439.742,340.617,175.563,49.662,160.479
C08534=1025.847,439.499,340.670,175.546,49.658,160.475
C08535=1025.834,439.255,340.723,175.528,49.653,160.470
C08536=1025.820,439.011,340.775,175.510,49.649,160.466
C08537=1025.807,438.767,340.827,175.492,49.645,160.462
C08538=1025.794,438.522,340.880,175.475,49.640,160.458
C08539=1025.780,438.279,340.933,175.457,49.636,160.454
C08540=1025.766,438.034,340.985,175.440,49.632,160.450
C08541=1025.752,437.789,341.037,175.423,49.628,160.446
C08542=1025.739,437.545,341.090,175.405,49.624,160.442
C08543=1025.726,437.301,341.142,175.388,49.620,160.437
C08544=1025.712,437.057,341.194,175.370,49.616,160.433
C08545=1025.699,436.813,341.246,175.354,49.611,160.429
C08546=1025.686,436.569,341.298,175.336,49.608,160.425
C08547=1025.673,436.324,341.350,175.319,49.603,160.421
C08548=1025.659,436.080,341.402,175.302,49.599,160.417
C08549=1025.646,435.836,341.453,175.285,49.595,160.414
C08550=1025.633,435.592,341.504,175.268,49.591,160.409
C08551=1025.620,435.347,341.557,175.251,49.587,160.406
C08552=1025.607,435.103,341.609,175.235,49.583,160.402
C08553=1025.594,434.858,341.660,175.218,49.579,160.398
C08554=1025.581,434.614,341.711,175.201,49.575,160.394
C08555=1025.568,434.369,341.762,175.185,49.571,160.390
C08556=1025.555,434.126,341.814,175.168,49.568,160.386
C08557=1025.542,433.881,341.866,175.152,49.564,160.383
C08558=1025.529,433.636,341.917,175.136,49.560,160.379
C08559=1025.516,433.392,341.968,175.119,49.556,160.375
C08560=1025.503,433.148,342.019,175.102,49.552,160.371
C08561=1025.490,432.903,342.070,175.086,49.549,160.368
C08562=1025.478,432.659,342.121,175.070,49.544,160.364
C08563=1025.464,432.414,342.172,175.054,49.540,160.360
C08564=1025.452,432.170,342.223,175.038,49.537,160.356
C08565=1025.439,431.924,342.274,175.022,49.533,160.353
C08566=1025.426,431.680,342.325,175.006,49.530,160.349
C08567=1025.414,431.436,342.375,174.990,49.525,160.345
C08568=1025.401,431.192,342.426,174.974,49.522,160.342
C08569=1025.387,430.946,342.476,174.958,49.518,160.338
C08570=1025.375,430.702,342.527,174.943,49.515,160.335
C08571=1025.362,430.457,342.577,174.926,49.511,160.331
C08572=1025.350,430.213,342.628,174.911,49.507,160.327
C08573=1025.337,429.968,342.678,174.895,49.504,160.324
C08574=1025.325,429.724,342.729,174.880,49.500,160.320
C08575=1025.313,429.479,342.779,174.864,49.497,160.317
C08576=1025.300,429.234,342.829,174.849,49.494,160.313
C08577=1025.288,428.990,342.879,174.833,49.490,160.310
C08578=1025.275,428.745,342.930,174.818,49.486,160.306
C08579=1025.263,428.501,342.980,174.802,49.483,160.303
C08580=1025.251,428.256,343.030,174.787,49.480,160.299
C08581=1025.238,428.011,343.080,174.772,49.476,160.296
C08582=1025.226,427.766,343.130,174.756,49.472,160.292
C08583=1025.214,427.521,343.180,174.742,49.469,160.289
C08584=1025.201,427.278,343.229,174.726,49.465,160.285
C08585=1025.189,427.032,343.279,174.712,49.462,160.282
C08586=1025.177,426.787,343.329,174.696,49.459,160.279
C08587=1025.165,426.542,343.379,174.681,49.455,160.275
C08588=1025.149,426.217,343.445,174.662,49.451,160.271
C08589=1025.133,425.891,343.511,174.642,49.446,160.266
C08590=1025.117,425.565,343.577,174.623,49.442,160.262
C08591=1025.101,425.239,343.642,174.603,49.438,160.258
C08592=1025.089,424.994,343.691,174.588,49.434,160.254
C08593=1025.077,424.748,343.741,174.573,49.431,160.251
C08594=1025.065,424.505,343.790,174.559,49.428,160.248
C08595=1025.053,424.259,343.839,174.545,49.425,160.245
C08596=1025.041,424.014,343.888,174.530,49.421,160.241
C08597=1025.029,423.769,343.938,174.516,49.418,160.238
C08598=1025.017,423.525,343.986,174.501,49.416,160.235
C08599=1025.005,423.279,344.035,174.486,49.412,160.232
C08600=1024.994,423.034,344.084,174.472,49.409,160.229
C08601=1024.982,422.790,344.133,174.458,49.406,160.225
C08602=1024.970,422.545,344.182,174.444,49.403,160.222
C08603=1024.958,422.299,344.231,174.429,49.400,160.219
C08604=1024.941,421.925,344.305,174.408,49.395,160.214
C08605=1024.923,421.551,344.379,174.387,49.390,160.210
C08606=1024.905,421.176,344.453,174.366,49.386,160.205
C08607=1024.887,420.802,344.527,174.344,49.381,160.200
C08608=1024.875,420.557,344.575,174.330,49.378,160.197
C08609=1024.864,420.313,344.624,174.316,49.375,160.194
C08610=1024.852,420.068,344.672,174.302,49.372,160.191
C08611=1024.841,419.822,344.720,174.289,49.370,160.188
C08612=1024.829,419.577,344.768,174.275,49.367,160.185
C08613=1024.818,419.332,344.816,174.262,49.364,160.182
C08614=1024.806,419.087,344.864,174.247,49.361,160.179
C08615=1024.795,418.841,344.912,174.234,49.359,160.177
C08616=1024.783,418.596,344.960,174.221,49.355,160.174
C08617=1024.772,418.351,345.008,174.207,49.353,160.171
C08618=1024.760,418.106,345.056,174.193,49.350,160.168
C08619=1024.749,417.861,345.103,174.180,49.347,160.165
C08620=1024.738,417.616,345.151,174.166,49.345,160.162
C08621=1024.727,417.371,345.199,174.154,49.342,160.159
C08622=1024.715,417.125,345.246,174.140,49.339,160.156
C08623=1024.704,416.880,345.294,174.127,49.336,160.153
C08624=1024.693,416.635,345.342,174.113,49.334,160.150
C08625=1024.682,416.389,345.390,174.101,49.331,160.148
C08626=1024.671,416.145,345.437,174.087,49.329,160.145
C08627=1024.660,415.899,345.485,174.074,49.325,160.142
C08628=1024.648,415.654,345.532,174.061,49.323,160.139
C08629=1024.637,415.409,345.579,174.048,49.320,160.136
C08630=1024.626,415.163,345.626,174.035,49.318,160.134
C08631=1024.614,414.918,345.674,174.022,49.316,160.131
C08632=1024.604,414.673,345.721,174.009,49.313,160.128
C08633=1024.592,414.427,345.768,173.996,49.310,160.125
C08634=1024.582,414.182,345.815,173.983,49.308,160.123
C08635=1024.570,413.936,345.862,173.971,49.306,160.120
C08636=1024.559,413.691,345.909,173.958,49.303,160.117
C08637=1024.548,413.446,345.956,173.945,49.300,160.115
C08638=1024.538,413.200,346.003,173.932,49.298,160.112
C08639=1024.527,412.955,346.049,173.919,49.296,160.109
C08640=1024.515,412.710,346.096,173.907,49.293,160.107
C08641=1024.504,412.465,346.143,173.894,49.291,160.104
C08642=1024.494,412.219,346.190,173.882,49.288,160.101
C08643=1024.483,411.974,346.236,173.869,49.286,160.099
C08644=1024.473,411.758,346.277,173.858,49.284,160.096
C08645=1024.464,411.542,346.319,173.848,49.282,160.094
C08646=1024.454,411.327,346.359,173.837,49.280,160.092
C08647=1024.445,411.112,346.400,173.826,49.278,160.090
C08648=1024.436,410.896,346.441,173.815,49.276,160.087
C08649=1024.426,410.681,346.482,173.804,49.274,160.085
C08650=1024.416,410.465,346.522,173.793,49.272,160.083
C08651=1024.408,410.249,346.563,173.782,49.270,160.081
C08652=1024.397,410.004,346.609,173.770,49.268,160.078
C08653=1024.386,409.759,346.656,173.757,49.265,160.075
C08654=1024.375,409.513,346.702,173.745,49.263,160.073
C08655=1024.365,409.267,346.748,173.733,49.261,160.070
C08656=1024.354,409.022,346.793,173.722,49.258,160.068
C08657=1024.343,408.776,346.839,173.709,49.256,160.065
C08658=1024.333,408.531,346.886,173.697,49.255,160.063
C08659=1024.322,408.286,346.932,173.685,49.252,160.060
C08660=1024.312,408.039,346.977,173.673,49.250,160.058
C08661=1024.301,407.794,347.023,173.661,49.248,160.056
C08662=1024.290,407.548,347.069,173.649,49.246,160.053
C08663=1024.280,407.303,347.114,173.638,49.244,160.051
C08664=1024.269,407.058,347.160,173.625,49.242,160.048
C08665=1024.258,406.812,347.206,173.614,49.240,160.046
C08666=1024.248,406.566,347.251,173.601,49.238,160.043
C08667=1024.237,406.321,347.297,173.590,49.236,160.041
C08668=1024.227,406.076,347.342,173.578,49.234,160.039
C08669=1024.217,405.830,347.387,173.566,49.232,160.036
C08670=1024.206,405.584,347.433,173.555,49.230,160.034
C08671=1024.196,405.339,347.479,173.543,49.228,160.032
C08672=1024.186,405.093,347.524,173.531,49.226,160.029
C08673=1024.175,404.847,347.570,173.520,49.224,160.027
C08674=1024.165,404.602,347.614,173.508,49.222,160.025
C08675=1024.155,404.356,347.659,173.496,49.221,160.022
C08676=1024.145,404.111,347.705,173.485,49.219,160.020
C08677=1024.134,403.865,347.750,173.474,49.217,160.018
C08678=1024.125,403.619,347.795,173.463,49.215,160.016
C08679=1024.114,403.374,347.841,173.451,49.213,160.013
C08680=1024.104,403.128,347.886,173.440,49.211,160.011
C08681=1024.094,402.882,347.931,173.428,49.209,160.009
C08682=1024.084,402.636,347.976,173.417,49.207,160.006
C08683=1024.074,402.391,348.020,173.405,49.206,160.004
C08684=1024.064,402.145,348.065,173.395,49.204,160.002
C08685=1024.054,401.899,348.110,173.384,49.202,160.000
C08686=1024.044,401.654,348.155,173.372,49.200,159.997
C08687=1024.034,401.408,348.200,173.361,49.198,159.995
C08688=1024.024,401.162,348.245,173.349,49.197,159.993
C08689=1024.014,400.917,348.290,173.338,49.195,159.991
C08690=1024.004,400.672,348.334,173.328,49.194,159.989
C08691=1023.994,400.425,348.379,173.316,49.192,159.986
C08692=1023.984,400.179,348.423,173.305,49.190,159.984
C08693=1023.974,399.934,348.467,173.294,49.188,159.982
C08694=1023.964,399.688,348.512,173.283,49.187,159.980
C08695=1023.955,399.442,348.556,173.272,49.186,159.978
C08696=1023.944,399.197,348.601,173.261,49.184,159.976
C08697=1023.934,398.950,348.645,173.251,49.182,159.974
C08698=1023.924,398.705,348.690,173.239,49.181,159.972
C08699=1023.914,398.459,348.733,173.229,49.180,159.970
C08700=1023.905,398.213,348.777,173.218,49.177,159.967
C08701=1023.895,397.967,348.822,173.207,49.176,159.965
C08702=1023.885,397.721,348.866,173.196,49.175,159.963
C08703=1023.876,397.475,348.910,173.185,49.173,159.961
C08704=1023.865,397.230,348.953,173.175,49.172,159.959
C08705=1023.856,396.984,348.998,173.164,49.170,159.957
C08706=1023.846,396.738,349.042,173.154,49.169,159.955
C08707=1023.836,396.492,349.086,173.143,49.167,159.953
C08708=1023.824,396.200,349.137,173.130,49.166,159.951
C08709=1023.813,395.907,349.189,173.117,49.164,159.948
C08710=1023.801,395.614,349.241,173.105,49.163,159.946
C08711=1023.790,395.322,349.294,173.093,49.161,159.944
C08712=1023.780,395.075,349.337,173.082,49.160,159.942
C08713=1023.770,394.829,349.381,173.072,49.159,159.940
C08714=1023.761,394.584,349.424,173.061,49.157,159.938
C08715=1023.752,394.338,349.468,173.051,49.156,159.936
C08716=1023.741,394.092,349.512,173.041,49.155,159.934
C08717=1023.732,393.846,349.555,173.030,49.153,159.932
C08718=1023.723,393.600,349.598,173.020,49.152,159.930
C08719=1023.713,393.354,349.642,173.009,49.151,159.928
C08720=1023.703,393.108,349.685,172.999,49.150,159.926
C08721=1023.694,392.863,349.728,172.989,49.148,159.924
C08722=1023.685,392.616,349.772,172.978,49.147,159.922
C08723=1023.675,392.370,349.815,172.968,49.146,159.920
C08724=1023.665,392.124,349.858,172.959,49.145,159.918
C08725=1023.656,391.878,349.901,172.949,49.144,159.917
C08726=1023.647,391.632,349.944,172.938,49.143,159.915
C08727=1023.637,391.386,349.987,172.928,49.142,159.913
C08728=1023.627,391.140,350.030,172.918,49.140,159.911
C08729=1023.619,390.894,350.073,172.908,49.139,159.909
C08730=1023.608,390.648,350.116,172.897,49.138,159.907
C08731=1023.599,390.402,350.159,172.888,49.137,159.906
C08732=1023.590,390.155,350.202,172.878,49.136,159.904
C08733=1023.581,389.909,350.245,172.868,49.135,159.902
C08734=1023.572,389.664,350.287,172.858,49.134,159.900
C08735=1023.562,389.417,350.330,172.848,49.133,159.898
C08736=1023.553,389.171,350.373,172.838,49.132,159.896
C08737=1023.543,388.925,350.416,172.828,49.131,159.895
C08738=1023.534,388.679,350.458,172.818,49.130,159.893
C08739=1023.525,388.433,350.501,172.808,49.130,159.891
C08740=1023.515,388.187,350.543,172.799,49.128,159.889
C08741=1023.507,387.940,350.586,172.789,49.127,159.888
C08742=1023.498,387.694,350.628,172.779,49.126,159.886
C08743=1023.488,387.448,350.671,172.770,49.126,159.884
C08744=1023.479,387.202,350.713,172.760,49.125,159.882
C08745=1023.470,386.956,350.755,172.750,49.124,159.881
C08746=1023.460,386.710,350.797,172.741,49.123,159.879
C08747=1023.451,386.463,350.840,172.731,49.122,159.877
C08748=1023.442,386.217,350.883,172.721,49.122,159.876
C08749=1023.433,385.971,350.924,172.712,49.120,159.874
C08750=1023.424,385.725,350.967,172.702,49.120,159.872
C08751=1023.415,385.479,351.008,172.693,49.119,159.870
C08752=1023.405,385.232,351.051,172.683,49.118,159.869
C08753=1023.396,384.986,351.092,172.673,49.117,159.867
C08754=1023.387,384.740,351.134,172.664,49.117,159.866
C08755=1023.378,384.493,351.176,172.654,49.116,159.864
C08756=1023.369,384.248,351.218,172.645,49.115,159.862
C08757=1023.360,384.001,351.260,172.635,49.114,159.861
C08758=1023.351,383.755,351.302,172.626,49.114,159.859
C08759=1023.342,383.508,351.343,172.616,49.113,159.857
C08760=1023.332,383.262,351.384,172.608,49.113,159.856
C08761=1023.323,383.016,351.426,172.598,49.112,159.854
C08762=1023.314,382.770,351.468,172.589,49.111,159.853
C08763=1023.305,382.523,351.510,172.579,49.111,159.851
C08764=1023.296,382.277,351.551,172.570,49.110,159.849
C08765=1023.288,382.031,351.593,172.560,49.109,159.848
C08766=1023.279,381.784,351.635,172.551,49.109,159.846
C08767=1023.269,381.538,351.676,172.542,49.109,159.845
C08768=1023.260,381.282,351.719,172.533,49.107,159.843
C08769=1023.251,381.026,351.762,172.523,49.107,159.841
C08770=1023.242,380.771,351.805,172.513,49.107,159.840
C08771=1023.233,380.515,351.848,172.504,49.106,159.838
C08772=1023.224,380.268,351.890,172.494,49.106,159.837
C08773=1023.215,380.022,351.930,172.486,49.105,159.835
C08774=1023.206,379.775,351.972,172.477,49.105,159.834
C08775=1023.197,379.529,352.014,172.467,49.104,159.832
C08776=1023.189,379.283,352.054,172.459,49.104,159.831
C08777=1023.180,379.036,352.096,172.450,49.103,159.829
C08778=1023.171,378.789,352.137,172.440,49.103,159.828
C08779=1023.163,378.544,352.178,172.432,49.102,159.826
C08780=1023.154,378.297,352.219,172.423,49.102,159.825
C08781=1023.145,378.051,352.260,172.413,49.102,159.823
C08782=1023.137,377.804,352.301,172.405,49.102,159.822
C08783=1023.128,377.558,352.343,172.396,49.101,159.820
C08784=1023.119,377.311,352.384,172.388,49.101,159.819
C08785=1023.111,377.065,352.424,172.378,49.100,159.817
C08786=1023.102,376.818,352.466,172.369,49.100,159.816
C08787=1023.093,376.572,352.506,172.361,49.099,159.814
C08788=1023.085,376.325,352.547,172.352,49.099,159.813
C08789=1023.076,376.078,352.588,172.342,49.099,159.811
C08790=1023.067,375.832,352.628,172.334,49.099,159.810
C08791=1023.059,375.585,352.669,172.325,49.098,159.809
C08792=1023.050,375.340,352.709,172.317,49.098,159.807
C08793=1023.041,375.093,352.750,172.308,49.098,159.806
C08794=1023.033,374.847,352.790,172.299,49.098,159.804
C08795=1023.024,374.600,352.831,172.290,49.098,159.803
C08796=1023.015,374.354,352.871,172.282,49.097,159.802
C08797=1023.007,374.107,352.912,172.273,49.097,159.800
C08798=1022.998,373.861,352.952,172.265,49.097,159.799
C08799=1022.989,373.613,352.993,172.256,49.097,159.798
C08800=1022.981,373.367,353.033,172.247,49.097,159.796
C08801=1022.973,373.121,353.073,172.238,49.097,159.795
C08802=1022.963,372.874,353.114,172.230,49.097,159.794
C08803=1022.956,372.627,353.154,172.222,49.097,159.792
C08804=1022.947,372.381,353.194,172.213,49.096,159.791
C08805=1022.939,372.134,353.234,172.205,49.096,159.790
C08806=1022.930,371.887,353.275,172.196,49.096,159.788
C08807=1022.922,371.641,353.315,172.188,49.096,159.787
C08808=1022.913,371.394,353.355,172.179,49.096,159.786
C08809=1022.905,371.148,353.395,172.171,49.096,159.784
C08810=1022.897,370.901,353.435,172.163,49.096,159.783
C08811=1022.888,370.655,353.475,172.154,49.096,159.782
C08812=1022.880,370.408,353.515,172.146,49.096,159.780
C08813=1022.871,370.161,353.555,172.138,49.096,159.779
C08814=1022.863,369.914,353.595,172.129,49.096,159.778
C08815=1022.855,369.668,353.634,172.121,49.096,159.777
C08816=1022.847,369.422,353.675,172.113,49.096,159.776
C08817=1022.838,369.175,353.714,172.104,49.096,159.774
C08818=1022.831,368.928,353.754,172.096,49.096,159.773
C08819=1022.822,368.681,353.794,172.088,49.096,159.772
C08820=1022.814,368.434,353.835,172.079,49.096,159.770
C08821=1022.805,368.188,353.874,172.071,49.097,159.769
C08822=1022.797,367.941,353.913,172.063,49.097,159.768
C08823=1022.789,367.694,353.953,172.055,49.097,159.767
C08824=1022.780,367.454,353.991,172.047,49.097,159.766
C08825=1022.772,367.214,354.030,172.038,49.097,159.764
C08826=1022.765,366.973,354.068,172.031,49.097,159.763
C08827=1022.756,366.734,354.107,172.023,49.098,159.762
C08828=1022.748,366.493,354.145,172.015,49.098,159.761
C08829=1022.740,366.253,354.183,172.007,49.099,159.760
C08830=1022.732,366.013,354.221,171.999,49.098,159.759
C08831=1022.724,365.772,354.259,171.991,49.099,159.757
C08832=1022.716,365.526,354.299,171.983,49.099,159.756
C08833=1022.708,365.279,354.337,171.975,49.099,159.755
C08834=1022.700,365.032,354.377,171.967,49.100,159.754
C08835=1022.691,364.785,354.417,171.959,49.100,159.753
C08836=1022.683,364.539,354.456,171.951,49.100,159.752
C08837=1022.675,364.291,354.495,171.943,49.100,159.750
C08838=1022.666,364.045,354.534,171.935,49.101,159.749
C08839=1022.658,363.798,354.572,171.927,49.101,159.748
C08840=1022.651,363.551,354.612,171.919,49.101,159.747
C08841=1022.643,363.305,354.651,171.911,49.102,159.746
C08842=1022.634,363.058,354.690,171.904,49.102,159.745
C08843=1022.626,362.811,354.729,171.896,49.102,159.744
C08844=1022.618,362.564,354.768,171.888,49.103,159.743
C08845=1022.610,362.317,354.806,171.880,49.103,159.741
C08846=1022.603,362.070,354.846,171.872,49.104,159.741
C08847=1022.594,361.823,354.885,171.865,49.104,159.739
C08848=1022.586,361.576,354.924,171.857,49.105,159.738
C08849=1022.578,361.330,354.962,171.849,49.105,159.737
C08850=1022.570,361.083,355.001,171.841,49.106,159.736
C08851=1022.562,360.836,355.040,171.833,49.106,159.735
C08852=1022.555,360.589,355.079,171.826,49.107,159.734
C08853=1022.547,360.342,355.118,171.818,49.107,159.733
C08854=1022.539,360.095,355.156,171.810,49.107,159.732
C08855=1022.531,359.849,355.195,171.802,49.108,159.731
C08856=1022.523,359.602,355.234,171.795,49.109,159.730
C08857=1022.515,359.355,355.272,171.787,49.109,159.729
C08858=1022.507,359.108,355.311,171.780,49.110,159.728
C08859=1022.499,358.861,355.349,171.772,49.110,159.727
C08860=1022.491,358.614,355.387,171.764,49.111,159.726
C08861=1022.482,358.367,355.425,171.757,49.111,159.725
C08862=1022.475,358.121,355.464,171.749,49.112,159.724
C08863=1022.467,357.873,355.502,171.741,49.113,159.723
C08864=1022.459,357.627,355.540,171.734,49.114,159.722
C08865=1022.451,357.379,355.578,171.726,49.114,159.721
C08866=1022.443,357.132,355.617,171.719,49.115,159.720
C08867=1022.436,356.886,355.655,171.711,49.115,159.719
C08868=1022.428,356.638,355.693,171.704,49.116,159.718
C08869=1022.419,356.392,355.731,171.696,49.117,159.717
C08870=1022.412,356.145,355.769,171.689,49.117,159.716
C08871=1022.404,355.898,355.808,171.681,49.118,159.715
C08872=1022.396,355.651,355.845,171.673,49.119,159.714
C08873=1022.388,355.404,355.884,171.667,49.120,159.713
C08874=1022.381,355.156,355.921,171.659,49.120,159.712
C08875=1022.373,354.910,355.959,171.652,49.121,159.711
C08876=1022.365,354.663,355.998,171.644,49.122,159.710
C08877=1022.357,354.416,356.035,171.636,49.123,159.709
C08878=1022.349,354.169,356.074,171.630,49.124,159.708
C08879=1022.341,353.922,356.111,171.622,49.125,159.707
C08880=1022.334,353.675,356.148,171.615,49.126,159.706
C08881=1022.326,353.427,356.187,171.607,49.126,159.705
C08882=1022.318,353.181,356.224,171.599,49.127,159.704
C08883=1022.311,352.933,356.261,171.593,49.128,159.703
C08884=1022.303,352.696,356.298,171.585,49.129,159.703
C08885=1022.295,352.460,356.333,171.578,49.130,159.702
C08886=1022.288,352.223,356.370,171.572,49.131,159.701
C08887=1022.281,351.986,356.406,171.565,49.131,159.700
C08888=1022.274,351.750,356.442,171.557,49.132,159.699
C08889=1022.265,351.512,356.478,171.550,49.133,159.698
C08890=1022.258,351.275,356.514,171.544,49.134,159.697
C08891=1022.251,351.039,356.550,171.537,49.135,159.697
C08892=1022.243,350.792,356.587,171.530,49.136,159.696
C08893=1022.236,350.545,356.624,171.523,49.137,159.695
C08894=1022.228,350.297,356.662,171.515,49.138,159.694
C08895=1022.220,350.050,356.699,171.508,49.139,159.693
C08896=1022.213,349.803,356.737,171.501,49.140,159.692
C08897=1022.206,349.556,356.774,171.494,49.141,159.691
C08898=1022.198,349.309,356.811,171.487,49.142,159.691
C08899=1022.190,349.062,356.849,171.480,49.143,159.690
C08900=1022.183,348.815,356.886,171.472,49.144,159.689
C08901=1022.175,348.568,356.923,171.466,49.145,159.688
C08902=1022.168,348.321,356.961,171.458,49.147,159.687
C08903=1022.160,348.074,356.998,171.452,49.147,159.686
C08904=1022.153,347.827,357.035,171.444,49.148,159.686
C08905=1022.145,347.579,357.071,171.437,49.150,159.685
C08906=1022.138,347.332,357.109,171.430,49.151,159.684
C08907=1022.130,347.086,357.146,171.423,49.152,159.683
C08908=1022.123,346.838,357.183,171.416,49.153,159.682
C08909=1022.115,346.591,357.220,171.409,49.154,159.682
C08910=1022.107,346.344,357.257,171.402,49.155,159.681
C08911=1022.100,346.096,357.293,171.395,49.157,159.680
C08912=1022.092,345.850,357.330,171.389,49.158,159.679
C08913=1022.084,345.602,357.367,171.381,49.159,159.678
C08914=1022.077,345.355,357.404,171.375,49.160,159.678
C08915=1022.069,345.108,357.440,171.367,49.162,159.677
C08916=1022.062,344.860,357.478,171.360,49.163,159.676
C08917=1022.054,344.613,357.514,171.354,49.164,159.675
C08918=1022.046,344.366,357.551,171.347,49.166,159.675
C08919=1022.040,344.118,357.588,171.340,49.166,159.674
C08920=1022.032,343.872,357.625,171.333,49.168,159.673
C08921=1022.024,343.625,357.661,171.326,49.169,159.672
C08922=1022.018,343.377,357.697,171.320,49.171,159.672
C08923=1022.010,343.130,357.734,171.312,49.172,159.671
C08924=1022.002,342.883,357.771,171.306,49.173,159.670
C08925=1021.995,342.635,357.807,171.299,49.174,159.670
C08926=1021.987,342.388,357.844,171.292,49.176,159.669
C08927=1021.980,342.141,357.880,171.285,49.177,159.668
C08928=1021.973,341.894,357.917,171.279,49.178,159.667
C08929=1021.965,341.646,357.953,171.272,49.180,159.667
C08930=1021.958,341.399,357.989,171.265,49.181,159.666
C08931=1021.950,341.153,358.026,171.259,49.183,159.665
C08932=1021.943,340.905,358.063,171.252,49.184,159.665
C08933=1021.936,340.657,358.099,171.245,49.186,159.664
C08934=1021.929,340.411,358.135,171.239,49.187,159.663
C08935=1021.921,340.163,358.171,171.231,49.189,159.663
C08936=1021.914,339.916,358.208,171.225,49.190,159.662
C08937=1021.907,339.669,358.244,171.219,49.191,159.661
C08938=1021.899,339.421,358.280,171.211,49.193,159.660
C08939=1021.891,339.174,358.316,171.205,49.194,159.660
C08940=1021.884,338.927,358.352,171.198,49.196,159.659
C08941=1021.877,338.679,358.387,171.191,49.197,159.658
C08942=1021.869,338.432,358.424,171.185,49.199,159.658
C08943=1021.862,338.185,358.460,171.179,49.200,159.657
C08944=1021.855,337.946,358.494,171.172,49.202,159.657
C08945=1021.848,337.709,358.529,171.166,49.204,159.656
C08946=1021.841,337.470,358.563,171.159,49.205,159.655
C08947=1021.835,337.231,358.598,171.152,49.207,159.655
C08948=1021.827,336.993,358.633,171.146,49.209,159.654
C08949=1021.820,336.754,358.667,171.140,49.210,159.654
C08950=1021.813,336.516,358.702,171.134,49.211,159.653
C08951=1021.806,336.277,358.736,171.128,49.213,159.652
C08952=1021.799,336.030,358.772,171.121,49.214,159.652
C08953=1021.791,335.783,358.808,171.115,49.216,159.651
C08954=1021.784,335.536,358.843,171.108,49.218,159.651
C08955=1021.777,335.288,358.879,171.101,49.219,159.650
C08956=1021.770,335.041,358.914,171.095,49.221,159.649
C08957=1021.762,334.793,358.951,171.089,49.223,159.649
C08958=1021.755,334.546,358.986,171.082,49.225,159.648
C08959=1021.748,334.299,359.022,171.076,49.226,159.647
C08960=1021.741,334.051,359.057,171.070,49.228,159.647
C08961=1021.734,333.804,359.093,171.063,49.229,159.646
C08962=1021.727,333.556,359.129,171.057,49.231,159.646
C08963=1021.719,333.310,359.164,171.050,49.233,159.645
C08964=1021.713,333.062,359.200,171.044,49.235,159.645
C08965=1021.705,332.814,359.235,171.038,49.237,159.644
C08966=1021.699,332.567,359.270,171.031,49.238,159.643
C08967=1021.691,332.320,359.306,171.024,49.240,159.643
C08968=1021.683,332.072,359.341,171.018,49.242,159.642
C08969=1021.677,331.825,359.376,171.012,49.244,159.642
C08970=1021.670,331.578,359.411,171.006,49.246,159.641
C08971=1021.662,331.330,359.447,171.000,49.248,159.641
C08972=1021.655,331.082,359.481,170.993,49.250,159.640
C08973=1021.648,330.836,359.517,170.987,49.252,159.640
C08974=1021.641,330.588,359.552,170.980,49.253,159.639
C08975=1021.634,330.340,359.588,170.974,49.255,159.639
C08976=1021.626,330.093,359.622,170.968,49.257,159.638
C08977=1021.619,329.846,359.657,170.961,49.259,159.638
C08978=1021.613,329.599,359.693,170.955,49.261,159.637
C08979=1021.605,329.350,359.728,170.949,49.263,159.637
C08980=1021.598,329.103,359.763,170.943,49.265,159.636
C08981=1021.591,328.856,359.798,170.937,49.267,159.636
C08982=1021.584,328.609,359.833,170.930,49.269,159.635
C08983=1021.578,328.361,359.868,170.924,49.271,159.635
C08984=1021.570,328.113,359.902,170.918,49.272,159.634
C08985=1021.563,327.866,359.937,170.912,49.274,159.634
C08986=1021.556,327.618,359.972,170.906,49.276,159.633
C08987=1021.549,327.371,360.008,170.900,49.278,159.633
C08988=1021.542,327.124,360.042,170.894,49.280,159.632
C08989=1021.535,326.876,360.077,170.887,49.283,159.632
C08990=1021.529,326.628,360.112,170.881,49.285,159.631
C08991=1021.521,326.381,360.146,170.875,49.287,159.631
C08992=1021.514,326.134,360.181,170.869,49.289,159.630
C08993=1021.506,325.886,360.215,170.863,49.291,159.630
C08994=1021.499,325.639,360.250,170.856,49.294,159.630
C08995=1021.492,325.391,360.284,170.850,49.296,159.629
C08996=1021.484,325.144,360.318,170.844,49.298,159.629
C08997=1021.478,324.896,360.353,170.838,49.300,159.628
C08998=1021.470,324.649,360.387,170.832,49.302,159.628
C08999=1021.463,324.401,360.421,170.826,49.304,159.627
C09000=1021.457,324.153,360.456,170.819,49.306,159.627
C09001=1021.449,323.906,360.490,170.814,49.309,159.626
C09002=1021.442,323.658,360.524,170.808,49.311,159.626
C09003=1021.435,323.411,360.559,170.802,49.314,159.626
C09004=1021.428,323.170,360.592,170.796,49.315,159.625
C09005=1021.421,322.930,360.625,170.790,49.317,159.625
C09006=1021.414,322.689,360.658,170.784,49.320,159.624
C09007=1021.408,322.449,360.691,170.778,49.322,159.624
C09008=1021.401,322.208,360.725,170.773,49.325,159.624
C09009=1021.394,321.967,360.758,170.767,49.326,159.623
C09010=1021.387,321.727,360.791,170.761,49.329,159.623
C09011=1021.380,321.486,360.825,170.755,49.331,159.622
C09012=1021.373,321.239,360.858,170.749,49.334,159.622
C09013=1021.366,320.991,360.892,170.743,49.336,159.622
C09014=1021.360,320.743,360.927,170.737,49.338,159.621
C09015=1021.352,320.496,360.961,170.731,49.340,159.621
C09016=1021.345,320.248,360.995,170.726,49.343,159.621
C09017=1021.338,320.000,361.029,170.720,49.345,159.620
C09018=1021.331,319.753,361.063,170.713,49.347,159.620
C09019=1021.325,319.506,361.097,170.707,49.350,159.620
C09020=1021.317,319.258,361.130,170.701,49.352,159.619
C09021=1021.311,319.010,361.165,170.696,49.355,159.619
C09022=1021.304,318.762,361.199,170.690,49.357,159.619
C09023=1021.297,318.515,361.232,170.684,49.359,159.618
C09024=1021.291,318.267,361.267,170.678,49.362,159.618
C09025=1021.284,318.020,361.300,170.673,49.364,159.617
C09026=1021.276,317.772,361.334,170.667,49.367,159.617
C09027=1021.270,317.525,361.368,170.661,49.369,159.617
C09028=1021.263,317.277,361.402,170.655,49.371,159.616
C09029=1021.256,317.029,361.436,170.650,49.374,159.616
C09030=1021.249,316.782,361.470,170.644,49.377,159.616
C09031=1021.242,316.535,361.503,170.638,49.379,159.615
C09032=1021.236,316.287,361.538,170.632,49.381,159.615
C09033=1021.229,316.039,361.571,170.627,49.384,159.615
C09034=1021.222,315.792,361.604,170.620,49.387,159.614
C09035=1021.215,315.544,361.638,170.614,49.389,159.614
C09036=1021.209,315.297,361.672,170.609,49.392,159.614
C09037=1021.202,315.049,361.706,170.603,49.394,159.614
C09038=1021.195,314.801,361.740,170.597,49.396,159.613
C09039=1021.189,314.553,361.773,170.591,49.399,159.613
C09040=1021.182,314.306,361.807,170.585,49.401,159.613
C09041=1021.175,314.059,361.840,170.580,49.404,159.612
C09042=1021.168,313.811,361.874,170.574,49.407,159.612
C09043=1021.163,313.563,361.907,170.568,49.409,159.612
C09044=1021.156,313.315,361.941,170.563,49.412,159.611
C09045=1021.149,313.069,361.975,170.557,49.414,159.611
C09046=1021.142,312.820,362.008,170.551,49.417,159.611
C09047=1021.136,312.573,362.042,170.546,49.420,159.611
C09048=1021.129,312.325,362.076,170.540,49.422,159.610
C09049=1021.123,312.078,362.108,170.534,49.425,159.610
C09050=1021.115,311.830,362.142,170.529,49.427,159.610
C09051=1021.109,311.582,362.175,170.523,49.430,159.609
C09052=1021.103,311.334,362.209,170.517,49.433,159.609
C09053=1021.096,311.087,362.242,170.512,49.435,159.609
C09054=1021.090,310.840,362.276,170.506,49.438,159.609
C09055=1021.083,310.592,362.309,170.502,49.441,159.608
C09056=1021.077,310.344,362.343,170.496,49.443,159.608
C09057=1021.070,310.096,362.376,170.490,49.446,159.608
C09058=1021.064,309.849,362.409,170.485,49.448,159.608
C09059=1021.057,309.602,362.442,170.478,49.452,159.607
C09060=1021.050,309.353,362.475,170.473,49.455,159.607
C09061=1021.043,309.106,362.507,170.467,49.458,159.607
C09062=1021.036,308.858,362.540,170.462,49.460,159.607
C09063=1021.029,308.610,362.573,170.456,49.463,159.606
C09064=1021.023,308.372,362.604,170.451,49.466,159.606
C09065=1021.016,308.134,362.636,170.446,49.468,159.606
C09066=1021.009,307.896,362.667,170.441,49.472,159.606
C09067=1021.003,307.658,362.699,170.435,49.474,159.606
C09068=1020.996,307.420,362.730,170.429,49.477,159.606
C09069=1020.990,307.182,362.762,170.424,49.480,159.605
C09070=1020.984,306.944,362.793,170.419,49.482,159.605
C09071=1020.977,306.706,362.824,170.414,49.486,159.605
C09072=1020.970,306.459,362.856,170.409,49.488,159.605
C09073=1020.963,306.210,362.889,170.403,49.491,159.605
C09074=1020.956,305.963,362.921,170.398,49.495,159.605
C09075=1020.950,305.715,362.954,170.392,49.497,159.604
C09076=1020.943,305.467,362.987,170.387,49.501,159.604
C09077=1020.936,305.220,363.019,170.381,49.503,159.604
C09078=1020.930,304.972,363.052,170.376,49.506,159.604
C09079=1020.922,304.724,363.084,170.371,49.510,159.604
C09080=1020.916,304.476,363.117,170.365,49.512,159.603
C09081=1020.910,304.229,363.149,170.360,49.515,159.603
C09082=1020.903,303.981,363.182,170.354,49.519,159.603
C09083=1020.896,303.734,363.214,170.349,49.521,159.603
C09084=1020.889,303.485,363.246,170.343,49.525,159.603
C09085=1020.883,303.237,363.279,170.338,49.528,159.603
C09086=1020.876,302.990,363.312,170.333,49.531,159.603
C09087=1020.869,302.743,363.344,170.327,49.534,159.602
C09088=1020.863,302.494,363.376,170.322,49.537,159.602
C09089=1020.856,302.246,363.408,170.316,49.540,159.602
C09090=1020.849,301.999,363.441,170.311,49.543,159.602
C09091=1020.843,301.751,363.473,170.306,49.547,159.602
C09092=1020.836,301.503,363.505,170.300,49.549,159.602
C09093=1020.830,301.256,363.538,170.295,49.552,159.602
C09094=1020.823,301.008,363.569,170.290,49.556,159.602
C09095=1020.817,300.760,363.602,170.284,49.559,159.601
C09096=1020.810,300.512,363.635,170.279,49.562,159.601
C09097=1020.803,300.264,363.667,170.274,49.565,159.601
C09098=1020.797,300.016,363.699,170.268,49.568,159.601
C09099=1020.790,299.768,363.731,170.263,49.571,159.601
C09100=1020.784,299.521,363.764,170.257,49.575,159.601
C09101=1020.778,299.273,363.796,170.252,49.578,159.601
C09102=1020.771,299.025,363.828,170.247,49.581,159.601
C09103=1020.765,298.777,363.860,170.241,49.584,159.600
C09104=1020.758,298.530,363.892,170.236,49.588,159.600
C09105=1020.752,298.282,363.924,170.231,49.591,159.600
C09106=1020.745,298.034,363.956,170.225,49.594,159.600
